(*Channel_43*)
	aPage_Channel[43].PARAM_NAME := 'Channel_43_ENC04';
	aPage_Channel[43].PARAM_00   := 4;
	aPage_Channel[43].PARAM_01   := 400;
	aPage_Channel[43].PARAM_02   := 0;
	aPage_Channel[43].PARAM_03   := 0;
	aPage_Channel[43].PARAM_04   := 0;
	aPage_Channel[43].PARAM_05   := 0;
	aPage_Channel[43].PARAM_06   := 0;
	aPage_Channel[43].PARAM_07   := 0;
	aPage_Channel[43].PARAM_08   := 0;
	aPage_Channel[43].PARAM_09   := 4;
	aPage_Channel[43].PARAM_10   := 0;

(*Channel_44*)
	aPage_Channel[44].PARAM_NAME := 'Channel_44_ENC05';
	aPage_Channel[44].PARAM_00   := 4;
	aPage_Channel[44].PARAM_01   := 500;
	aPage_Channel[44].PARAM_02   := 0;
	aPage_Channel[44].PARAM_03   := 0;
	aPage_Channel[44].PARAM_04   := 0;
	aPage_Channel[44].PARAM_05   := 0;
	aPage_Channel[44].PARAM_06   := 0;
	aPage_Channel[44].PARAM_07   := 0;
	aPage_Channel[44].PARAM_08   := 0;
	aPage_Channel[44].PARAM_09   := 5;
	aPage_Channel[44].PARAM_10   := 0;

(*Channel_45*)
	aPage_Channel[45].PARAM_NAME := 'Channel_45_ENC06';
	aPage_Channel[45].PARAM_00   := 4;
	aPage_Channel[45].PARAM_01   := 600;
	aPage_Channel[45].PARAM_02   := 0;
	aPage_Channel[45].PARAM_03   := 0;
	aPage_Channel[45].PARAM_04   := 0;
	aPage_Channel[45].PARAM_05   := 0;
	aPage_Channel[45].PARAM_06   := 0;
	aPage_Channel[45].PARAM_07   := 0;
	aPage_Channel[45].PARAM_08   := 0;
	aPage_Channel[45].PARAM_09   := 6;
	aPage_Channel[45].PARAM_10   := 0;

(*Channel_46*)
	aPage_Channel[46].PARAM_NAME := 'Channel_46_ENC07';
	aPage_Channel[46].PARAM_00   := 4;
	aPage_Channel[46].PARAM_01   := 700;
	aPage_Channel[46].PARAM_02   := 0;
	aPage_Channel[46].PARAM_03   := 0;
	aPage_Channel[46].PARAM_04   := 0;
	aPage_Channel[46].PARAM_05   := 0;
	aPage_Channel[46].PARAM_06   := 0;
	aPage_Channel[46].PARAM_07   := 0;
	aPage_Channel[46].PARAM_08   := 0;
	aPage_Channel[46].PARAM_09   := 7;
	aPage_Channel[46].PARAM_10   := 0;

(*Channel_47*)
	aPage_Channel[47].PARAM_NAME := 'Channel_47_ENC08';
	aPage_Channel[47].PARAM_00   := 4;
	aPage_Channel[47].PARAM_01   := 800;
	aPage_Channel[47].PARAM_02   := 0;
	aPage_Channel[47].PARAM_03   := 0;
	aPage_Channel[47].PARAM_04   := 0;
	aPage_Channel[47].PARAM_05   := 0;
	aPage_Channel[47].PARAM_06   := 0;
	aPage_Channel[47].PARAM_07   := 0;
	aPage_Channel[47].PARAM_08   := 0;
	aPage_Channel[47].PARAM_09   := 8;
	aPage_Channel[47].PARAM_10   := 0;

(*Channel_48*)
	aPage_Channel[48].PARAM_NAME := 'Channel_48_FRM01';
	aPage_Channel[48].PARAM_00   := 5;
	aPage_Channel[48].PARAM_01   := 1;
	aPage_Channel[48].PARAM_02   := 2;
	aPage_Channel[48].PARAM_03   := 3;
	aPage_Channel[48].PARAM_04   := 4;
	aPage_Channel[48].PARAM_05   := 5;
	aPage_Channel[48].PARAM_06   := 0;
	aPage_Channel[48].PARAM_07   := 0;
	aPage_Channel[48].PARAM_08   := 0;
	aPage_Channel[48].PARAM_09   := 1;
	aPage_Channel[48].PARAM_10   := 0;

(*Channel_49*)
	aPage_Channel[49].PARAM_NAME := 'Channel_49_FRM02';
	aPage_Channel[49].PARAM_00   := 5;
	aPage_Channel[49].PARAM_01   := 1;
	aPage_Channel[49].PARAM_02   := 2;
	aPage_Channel[49].PARAM_03   := 3;
	aPage_Channel[49].PARAM_04   := 4;
	aPage_Channel[49].PARAM_05   := 5;
	aPage_Channel[49].PARAM_06   := 0;
	aPage_Channel[49].PARAM_07   := 0;
	aPage_Channel[49].PARAM_08   := 0;
	aPage_Channel[49].PARAM_09   := 2;
	aPage_Channel[49].PARAM_10   := 0;

(*Channel_50*)
	aPage_Channel[50].PARAM_NAME := 'Channel_50_FRM03';
	aPage_Channel[50].PARAM_00   := 5;
	aPage_Channel[50].PARAM_01   := 1;
	aPage_Channel[50].PARAM_02   := 2;
	aPage_Channel[50].PARAM_03   := 3;
	aPage_Channel[50].PARAM_04   := 4;
	aPage_Channel[50].PARAM_05   := 5;
	aPage_Channel[50].PARAM_06   := 0;
	aPage_Channel[50].PARAM_07   := 0;
	aPage_Channel[50].PARAM_08   := 0;
	aPage_Channel[50].PARAM_09   := 3;
	aPage_Channel[50].PARAM_10   := 0;

(*Channel_51*)
	aPage_Channel[51].PARAM_NAME := 'Channel_51_FRM04';
	aPage_Channel[51].PARAM_00   := 5;
	aPage_Channel[51].PARAM_01   := 1;
	aPage_Channel[51].PARAM_02   := 2;
	aPage_Channel[51].PARAM_03   := 3;
	aPage_Channel[51].PARAM_04   := 4;
	aPage_Channel[51].PARAM_05   := 5;
	aPage_Channel[51].PARAM_06   := 0;
	aPage_Channel[51].PARAM_07   := 0;
	aPage_Channel[51].PARAM_08   := 0;
	aPage_Channel[51].PARAM_09   := 4;
	aPage_Channel[51].PARAM_10   := 0;

(*Channel_52*)
	aPage_Channel[52].PARAM_NAME := 'Channel_52_FRM05';
	aPage_Channel[52].PARAM_00   := 5;
	aPage_Channel[52].PARAM_01   := 1;
	aPage_Channel[52].PARAM_02   := 2;
	aPage_Channel[52].PARAM_03   := 3;
	aPage_Channel[52].PARAM_04   := 4;
	aPage_Channel[52].PARAM_05   := 5;
	aPage_Channel[52].PARAM_06   := 0;
	aPage_Channel[52].PARAM_07   := 0;
	aPage_Channel[52].PARAM_08   := 0;
	aPage_Channel[52].PARAM_09   := 5;
	aPage_Channel[52].PARAM_10   := 0;

(*Channel_53*)
	aPage_Channel[53].PARAM_NAME := 'Channel_53_FRM06';
	aPage_Channel[53].PARAM_00   := 5;
	aPage_Channel[53].PARAM_01   := 1;
	aPage_Channel[53].PARAM_02   := 2;
	aPage_Channel[53].PARAM_03   := 3;
	aPage_Channel[53].PARAM_04   := 4;
	aPage_Channel[53].PARAM_05   := 5;
	aPage_Channel[53].PARAM_06   := 0;
	aPage_Channel[53].PARAM_07   := 0;
	aPage_Channel[53].PARAM_08   := 0;
	aPage_Channel[53].PARAM_09   := 6;
	aPage_Channel[53].PARAM_10   := 0;

(*Channel_54*)
	aPage_Channel[54].PARAM_NAME := 'Channel_54_FRM07';
	aPage_Channel[54].PARAM_00   := 5;
	aPage_Channel[54].PARAM_01   := 1;
	aPage_Channel[54].PARAM_02   := 2;
	aPage_Channel[54].PARAM_03   := 3;
	aPage_Channel[54].PARAM_04   := 4;
	aPage_Channel[54].PARAM_05   := 5;
	aPage_Channel[54].PARAM_06   := 0;
	aPage_Channel[54].PARAM_07   := 0;
	aPage_Channel[54].PARAM_08   := 0;
	aPage_Channel[54].PARAM_09   := 7;
	aPage_Channel[54].PARAM_10   := 0;

(*Channel_55*)
	aPage_Channel[55].PARAM_NAME := 'Channel_55_FRM08';
	aPage_Channel[55].PARAM_00   := 5;
	aPage_Channel[55].PARAM_01   := 1;
	aPage_Channel[55].PARAM_02   := 2;
	aPage_Channel[55].PARAM_03   := 3;
	aPage_Channel[55].PARAM_04   := 4;
	aPage_Channel[55].PARAM_05   := 5;
	aPage_Channel[55].PARAM_06   := 0;
	aPage_Channel[55].PARAM_07   := 0;
	aPage_Channel[55].PARAM_08   := 0;
	aPage_Channel[55].PARAM_09   := 8;
	aPage_Channel[55].PARAM_10   := 0;

(*Channel_56*)
	aPage_Channel[56].PARAM_NAME := 'Channel_56_SPR01';
	aPage_Channel[56].PARAM_00   := 6;
	aPage_Channel[56].PARAM_01   := 1;
	aPage_Channel[56].PARAM_02   := 1;
	aPage_Channel[56].PARAM_03   := 1;
	aPage_Channel[56].PARAM_04   := 1;
	aPage_Channel[56].PARAM_05   := 1;
	aPage_Channel[56].PARAM_06   := 0;
	aPage_Channel[56].PARAM_07   := 0;
	aPage_Channel[56].PARAM_08   := 0;
	aPage_Channel[56].PARAM_09   := 1;
	aPage_Channel[56].PARAM_10   := 0;

(*Channel_57*)
	aPage_Channel[57].PARAM_NAME := 'Channel_57_SPR02';
	aPage_Channel[57].PARAM_00   := 6;
	aPage_Channel[57].PARAM_01   := 1;
	aPage_Channel[57].PARAM_02   := 1;
	aPage_Channel[57].PARAM_03   := 1;
	aPage_Channel[57].PARAM_04   := 1;
	aPage_Channel[57].PARAM_05   := 1;
	aPage_Channel[57].PARAM_06   := 0;
	aPage_Channel[57].PARAM_07   := 0;
	aPage_Channel[57].PARAM_08   := 0;
	aPage_Channel[57].PARAM_09   := 2;
	aPage_Channel[57].PARAM_10   := 0;

(*Channel_58*)
	aPage_Channel[58].PARAM_NAME := 'Channel_58_SPR03';
	aPage_Channel[58].PARAM_00   := 6;
	aPage_Channel[58].PARAM_01   := 1;
	aPage_Channel[58].PARAM_02   := 1;
	aPage_Channel[58].PARAM_03   := 1;
	aPage_Channel[58].PARAM_04   := 1;
	aPage_Channel[58].PARAM_05   := 1;
	aPage_Channel[58].PARAM_06   := 0;
	aPage_Channel[58].PARAM_07   := 0;
	aPage_Channel[58].PARAM_08   := 0;
	aPage_Channel[58].PARAM_09   := 3;
	aPage_Channel[58].PARAM_10   := 0;

(*Channel_59*)
	aPage_Channel[59].PARAM_NAME := 'Channel_59_SPR04';
	aPage_Channel[59].PARAM_00   := 6;
	aPage_Channel[59].PARAM_01   := 1;
	aPage_Channel[59].PARAM_02   := 1;
	aPage_Channel[59].PARAM_03   := 1;
	aPage_Channel[59].PARAM_04   := 1;
	aPage_Channel[59].PARAM_05   := 1;
	aPage_Channel[59].PARAM_06   := 0;
	aPage_Channel[59].PARAM_07   := 0;
	aPage_Channel[59].PARAM_08   := 0;
	aPage_Channel[59].PARAM_09   := 4;
	aPage_Channel[59].PARAM_10   := 0;

(*Channel_60*)
	aPage_Channel[60].PARAM_NAME := 'Channel_60_SPR05';
	aPage_Channel[60].PARAM_00   := 6;
	aPage_Channel[60].PARAM_01   := 1;
	aPage_Channel[60].PARAM_02   := 1;
	aPage_Channel[60].PARAM_03   := 1;
	aPage_Channel[60].PARAM_04   := 1;
	aPage_Channel[60].PARAM_05   := 1;
	aPage_Channel[60].PARAM_06   := 0;
	aPage_Channel[60].PARAM_07   := 0;
	aPage_Channel[60].PARAM_08   := 0;
	aPage_Channel[60].PARAM_09   := 5;
	aPage_Channel[60].PARAM_10   := 0;

(*Channel_61*)
	aPage_Channel[61].PARAM_NAME := 'Channel_61_SPR06';
	aPage_Channel[61].PARAM_00   := 6;
	aPage_Channel[61].PARAM_01   := 1;
	aPage_Channel[61].PARAM_02   := 1;
	aPage_Channel[61].PARAM_03   := 1;
	aPage_Channel[61].PARAM_04   := 1;
	aPage_Channel[61].PARAM_05   := 1;
	aPage_Channel[61].PARAM_06   := 0;
	aPage_Channel[61].PARAM_07   := 0;
	aPage_Channel[61].PARAM_08   := 0;
	aPage_Channel[61].PARAM_09   := 6;
	aPage_Channel[61].PARAM_10   := 0;

(*Channel_62*)
	aPage_Channel[62].PARAM_NAME := 'Channel_62_SPR07';
	aPage_Channel[62].PARAM_00   := 6;
	aPage_Channel[62].PARAM_01   := 1;
	aPage_Channel[62].PARAM_02   := 1;
	aPage_Channel[62].PARAM_03   := 1;
	aPage_Channel[62].PARAM_04   := 1;
	aPage_Channel[62].PARAM_05   := 1;
	aPage_Channel[62].PARAM_06   := 0;
	aPage_Channel[62].PARAM_07   := 0;
	aPage_Channel[62].PARAM_08   := 0;
	aPage_Channel[62].PARAM_09   := 7;
	aPage_Channel[62].PARAM_10   := 0;

(*Channel_63*)
	aPage_Channel[63].PARAM_NAME := 'Channel_63_SPR08';
	aPage_Channel[63].PARAM_00   := 6;
	aPage_Channel[63].PARAM_01   := 1;
	aPage_Channel[63].PARAM_02   := 1;
	aPage_Channel[63].PARAM_03   := 1;
	aPage_Channel[63].PARAM_04   := 1;
	aPage_Channel[63].PARAM_05   := 1;
	aPage_Channel[63].PARAM_06   := 0;
	aPage_Channel[63].PARAM_07   := 0;
	aPage_Channel[63].PARAM_08   := 0;
	aPage_Channel[63].PARAM_09   := 8;
	aPage_Channel[63].PARAM_10   := 0;

(*-----------------------------------------------------------------------------------------------------------------------------------------------------------------------------------*)
(**)

	DefaultSettingsTestModeRecovery;

	bCurrModeChange := 0;

END_IF;
END_PROGRAM

(* POU Default_Settings/FLASH_TO_PAGE_CHANNEL, ST *)
FUNCTION_BLOCK FLASH_TO_PAGE_CHANNEL

VAR_INPUT
	bInit         : BOOL;
END_VAR

VAR_OUTPUT
END_VAR

VAR
	instFRAMWrite : FRAMWRITE;
	i             : INT := 0;
END_VAR
(*-----------------------------------------------------------------------------------------------------------------------------------------------------------------------------------*)
(*Запись в энергонезависимую память установочных параметров, коэффициентов*)

FOR i := 0 TO 63 DO
	instFRAMWrite(Enable := 1, DST := iMemAdrArrayParamName + i * 32, LEN := 32, SRC := ADR(aPage_Channel[i].PARAM_NAME));

	instFRAMWrite(Enable := 1, DST := iMemAdrArrayParam00 + i * 4,    LEN := 4,  SRC := ADR(aPage_Channel[i].PARAM_00));
	instFRAMWrite(Enable := 1, DST := iMemAdrArrayParam01 + i * 4,    LEN := 4,  SRC := ADR(aPage_Channel[i].PARAM_01));
	instFRAMWrite(Enable := 1, DST := iMemAdrArrayParam02 + i * 4,    LEN := 4,  SRC := ADR(aPage_Channel[i].PARAM_02));
	instFRAMWrite(Enable := 1, DST := iMemAdrArrayParam03 + i * 4,    LEN := 4,  SRC := ADR(aPage_Channel[i].PARAM_03));
	instFRAMWrite(Enable := 1, DST := iMemAdrArrayParam04 + i * 4,    LEN := 4,  SRC := ADR(aPage_Channel[i].PARAM_04));
	instFRAMWrite(Enable := 1, DST := iMemAdrArrayParam05 + i * 4,    LEN := 4,  SRC := ADR(aPage_Channel[i].PARAM_05));
	instFRAMWrite(Enable := 1, DST := iMemAdrArrayParam06 + i * 4,    LEN := 4,  SRC := ADR(aPage_Channel[i].PARAM_06));
	instFRAMWrite(Enable := 1, DST := iMemAdrArrayParam07 + i * 4,    LEN := 4,  SRC := ADR(aPage_Channel[i].PARAM_07));

	instFRAMWrite(Enable := 1, DST := iMemAdrArrayParam09 + i * 4,    LEN := 4,  SRC := ADR(aPage_Channel[i].PARAM_09));
	instFRAMWrite(Enable := 1, DST := iMemAdrArrayParam10 + i * 4,    LEN := 4,  SRC := ADR(aPage_Channel[i].PARAM_10));
END_FOR;
END_FUNCTION_BLOCK

(* POU Default_Settings/Default_Settings_UnitMode_processing, ST *)
PROGRAM Default_Settings_UnitMode_processing

VAR_INPUT
	bInit                           : BOOL;
END_VAR

VAR
	DefaultSettingsUnitModeRecovery : FLASH_TO_PAGE_CHANNEL;
END_VAR
(*-----------------------------------------------------------------------------------------------------------------------------------------------------------------------------------*)
(*Восстановление заводских установок*)

IF bCurrModeChange = 1 AND dwCurrMode = 1 THEN

(*Channel_00*)
	aPage_Channel[00].PARAM_NAME := 'Давл. подпитки';
	aPage_Channel[00].PARAM_00   := 0;
	aPage_Channel[00].PARAM_01   := 3259;
	aPage_Channel[00].PARAM_02   := 648;
	aPage_Channel[00].PARAM_03   := 1.6 (*1.378951*);(*МПа, = 200 PSI*)
	aPage_Channel[00].PARAM_04   := 0;
	aPage_Channel[00].PARAM_05   := 100;
	aPage_Channel[00].PARAM_06   := 0;
	aPage_Channel[00].PARAM_07   := 0;
	aPage_Channel[00].PARAM_08   := 0;
	aPage_Channel[00].PARAM_09   := 1;
	aPage_Channel[00].PARAM_10   := 0;

(*Channel_01*)
	aPage_Channel[01].PARAM_NAME := 'Темп. азота жидкого';
	aPage_Channel[01].PARAM_00   := 0;
	aPage_Channel[01].PARAM_01   := 3259;
	aPage_Channel[01].PARAM_02   := 648;
	aPage_Channel[01].PARAM_03   := 76.666667;(*C, = 170 F*)
	aPage_Channel[01].PARAM_04   :=-195.555556;(*C, = 320 F*)
	aPage_Channel[01].PARAM_05   := 100;
	aPage_Channel[01].PARAM_06   := 0;
	aPage_Channel[01].PARAM_07   := 0;
	aPage_Channel[01].PARAM_08   := 0;
	aPage_Channel[01].PARAM_09   := 2;
	aPage_Channel[01].PARAM_10   := 0;

(*Channel_02*)
	aPage_Channel[02].PARAM_NAME := 'Темп. нагнетания';
	aPage_Channel[02].PARAM_00   := 0;
	aPage_Channel[02].PARAM_01   := 3259;
	aPage_Channel[02].PARAM_02   := 648;
	aPage_Channel[02].PARAM_03   := 50;
	aPage_Channel[02].PARAM_04   :=-50;
	aPage_Channel[02].PARAM_05   := 100;
	aPage_Channel[02].PARAM_06   := 0;
	aPage_Channel[02].PARAM_07   := 0;
	aPage_Channel[02].PARAM_08   := 0;
	aPage_Channel[02].PARAM_09   := 4;
	aPage_Channel[02].PARAM_10   := 0;

(*Channel_03*)
	aPage_Channel[03].PARAM_NAME := 'Давл. нагнетания';
	aPage_Channel[03].PARAM_00   := 0;
	aPage_Channel[03].PARAM_01   := 3259;
	aPage_Channel[03].PARAM_02   := 648;
	aPage_Channel[03].PARAM_03   := 103.421351;(*МПа, = 15000 PSI*)
	aPage_Channel[03].PARAM_04   := 0;
	aPage_Channel[03].PARAM_05   := 100;
	aPage_Channel[03].PARAM_06   := 0;
	aPage_Channel[03].PARAM_07   := 0;
	aPage_Channel[03].PARAM_08   := 0;
	aPage_Channel[03].PARAM_09   := 5;
	aPage_Channel[03].PARAM_10   := 0;

(*Channel_04*)
	aPage_Channel[04].PARAM_NAME := 'Давл. гидронагрева';
	aPage_Channel[04].PARAM_00   := 0;
	aPage_Channel[04].PARAM_01   := 3259;
	aPage_Channel[04].PARAM_02   := 648;
	aPage_Channel[04].PARAM_03   := 40;
	aPage_Channel[04].PARAM_04   := 0;
	aPage_Channel[04].PARAM_05   := 100;
	aPage_Channel[04].PARAM_06   := 0;
	aPage_Channel[04].PARAM_07   := 0;
	aPage_Channel[04].PARAM_08   := 0;
	aPage_Channel[04].PARAM_09   := 6;
	aPage_Channel[04].PARAM_10   := 0;

(*Channel_05*)
	aPage_Channel[05].PARAM_NAME := 'Темп. ОЖ до испарителя';
	aPage_Channel[05].PARAM_00   := 0;
	aPage_Channel[05].PARAM_01   := 3259;
	aPage_Channel[05].PARAM_02   := 648;
	aPage_Channel[05].PARAM_03   := 150;
	aPage_Channel[05].PARAM_04   :=-50;
	aPage_Channel[05].PARAM_05   := 100;
	aPage_Channel[05].PARAM_06   := 0;
	aPage_Channel[05].PARAM_07   := 0;
	aPage_Channel[05].PARAM_08   := 0;
	aPage_Channel[05].PARAM_09   := 3;
	aPage_Channel[05].PARAM_10   := 0;

(*Channel_06*)
	aPage_Channel[06].PARAM_NAME := 'Обороты НВД';
	aPage_Channel[06].PARAM_00   := 1;
	aPage_Channel[06].PARAM_01   := 8_200;
	aPage_Channel[06].PARAM_02   := 0;
	aPage_Channel[06].PARAM_03   := 6_000;
	aPage_Channel[06].PARAM_04   := 0;
	aPage_Channel[06].PARAM_05   := 1_000;
	aPage_Channel[06].PARAM_06   := 0;
	aPage_Channel[06].PARAM_07   := 0;
	aPage_Channel[06].PARAM_08   := 0;
	aPage_Channel[06].PARAM_09   := 1;
	aPage_Channel[06].PARAM_10   := 0;

(*Channel_07*)
	aPage_Channel[07].PARAM_NAME := 'Давл. гидронагрева';
	aPage_Channel[07].PARAM_00   := 2;
	aPage_Channel[07].PARAM_01   := 100;
	aPage_Channel[07].PARAM_02   := 0;
	aPage_Channel[07].PARAM_03   := 540 (*500*);
	aPage_Channel[07].PARAM_04   := 0;
	aPage_Channel[07].PARAM_05   := 4_000;
	aPage_Channel[07].PARAM_06   := 0;
	aPage_Channel[07].PARAM_07   := 0;
	aPage_Channel[07].PARAM_08   := 0;
	aPage_Channel[07].PARAM_09   := 1;
	aPage_Channel[07].PARAM_10   := 0;

(*Channel_08*)
	aPage_Channel[08].PARAM_NAME := 'Обороты НВД';
	aPage_Channel[08].PARAM_00   := 2;
	aPage_Channel[08].PARAM_01   := 100;
	aPage_Channel[08].PARAM_02   := 0;
	aPage_Channel[08].PARAM_03   := 460 (*400*);
	aPage_Channel[08].PARAM_04   := 0;
	aPage_Channel[08].PARAM_05   := 4_000;
	aPage_Channel[08].PARAM_06   := 0;
	aPage_Channel[08].PARAM_07   := 0;
	aPage_Channel[08].PARAM_08   := 0;
	aPage_Channel[08].PARAM_09   := 2;
	aPage_Channel[08].PARAM_10   := 0;

(*Channel_09*)
	aPage_Channel[09].PARAM_NAME := 'Давл. подпитки';
	aPage_Channel[09].PARAM_00   := 2;
	aPage_Channel[09].PARAM_01   := 100;
	aPage_Channel[09].PARAM_02   := 0;
	aPage_Channel[09].PARAM_03   := 400;
	aPage_Channel[09].PARAM_04   := 0;
	aPage_Channel[09].PARAM_05   := 4_000;
	aPage_Channel[09].PARAM_06   := 0;
	aPage_Channel[09].PARAM_07   := 0;
	aPage_Channel[09].PARAM_08   := 0;
	aPage_Channel[09].PARAM_09   := 3;
	aPage_Channel[09].PARAM_10   := 0;

(*Channel_10*)
	aPage_Channel[10].PARAM_NAME := 'Давл. гидронагрева';
	aPage_Channel[10].PARAM_00   := 3;
	aPage_Channel[10].PARAM_01   := 20 (*250*);
	aPage_Channel[10].PARAM_02   := 50;
	aPage_Channel[10].PARAM_03   := 0;
	aPage_Channel[10].PARAM_04   := 0;
	aPage_Channel[10].PARAM_05   := 0;
	aPage_Channel[10].PARAM_06   := 0;
	aPage_Channel[10].PARAM_07   := 0;
	aPage_Channel[10].PARAM_08   := 0;
	aPage_Channel[10].PARAM_09   := 1;
	aPage_Channel[10].PARAM_10   := 0;

(*Channel_11*)
	aPage_Channel[11].PARAM_NAME := 'Обороты НВД';
	aPage_Channel[11].PARAM_00   := 3;
	aPage_Channel[11].PARAM_01   := 0.001 (*0.005*);
	aPage_Channel[11].PARAM_02   := 0.05;
	aPage_Channel[11].PARAM_03   := 0;
	aPage_Channel[11].PARAM_04   := 180;
	aPage_Channel[11].PARAM_05   := 0;
	aPage_Channel[11].PARAM_06   := 0;
	aPage_Channel[11].PARAM_07   := 0;
	aPage_Channel[11].PARAM_08   := 0;
	aPage_Channel[11].PARAM_09   := 2;
	aPage_Channel[11].PARAM_10   := 0;

(*Channel_12*)
	aPage_Channel[12].PARAM_NAME := 'Давл. подпитки';
	aPage_Channel[12].PARAM_00   := 3;
	aPage_Channel[12].PARAM_01   := 30 (*80*);
	aPage_Channel[12].PARAM_02   := 0.250;
	aPage_Channel[12].PARAM_03   := 0;
	aPage_Channel[12].PARAM_04   := 0;
	aPage_Channel[12].PARAM_05   := 0;
	aPage_Channel[12].PARAM_06   := 0;
	aPage_Channel[12].PARAM_07   := 0;
	aPage_Channel[12].PARAM_08   := 0;
	aPage_Channel[12].PARAM_09   := 3;
	aPage_Channel[12].PARAM_10   := 0;

(*Channel_13*)
	aPage_Channel[13].PARAM_NAME := 'Channel_13';
	aPage_Channel[13].PARAM_00   := 9;
	aPage_Channel[13].PARAM_01   := 1;
	aPage_Channel[13].PARAM_02   := 1;
	aPage_Channel[13].PARAM_03   := 1;
	aPage_Channel[13].PARAM_04   := 1;
	aPage_Channel[13].PARAM_05   := 1;
	aPage_Channel[13].PARAM_06   := 0;
	aPage_Channel[13].PARAM_07   := 0;
	aPage_Channel[13].PARAM_08   := 0;
	aPage_Channel[13].PARAM_09   := 0;
	aPage_Channel[13].PARAM_10   := 0;

(*Channel_14*)
	aPage_Channel[14].PARAM_NAME := 'Channel_14';
	aPage_Channel[14].PARAM_00   := 9;
	aPage_Channel[14].PARAM_01   := 1;
	aPage_Channel[14].PARAM_02   := 1;
	aPage_Channel[14].PARAM_03   := 1;
	aPage_Channel[14].PARAM_04   := 1;
	aPage_Channel[14].PARAM_05   := 1;
	aPage_Channel[14].PARAM_06   := 0;
	aPage_Channel[14].PARAM_07   := 0;
	aPage_Channel[14].PARAM_08   := 0;
	aPage_Channel[14].PARAM_09   := 0;
	aPage_Channel[14].PARAM_10   := 0;

(*Channel_15*)
	aPage_Channel[15].PARAM_NAME := 'Channel_15';
	aPage_Channel[15].PARAM_00   := 9;
	aPage_Channel[15].PARAM_01   := 1;
	aPage_Channel[15].PARAM_02   := 1;
	aPage_Channel[15].PARAM_03   := 1;
	aPage_Channel[15].PARAM_04   := 1;
	aPage_Channel[15].PARAM_05   := 1;
	aPage_Channel[15].PARAM_06   := 0;
	aPage_Channel[15].PARAM_07   := 0;
	aPage_Channel[15].PARAM_08   := 0;
	aPage_Channel[15].PARAM_09   := 0;
	aPage_Channel[15].PARAM_10   := 0;

(*Channel_16*)
	aPage_Channel[16].PARAM_NAME := 'Channel_16';
	aPage_Channel[16].PARAM_00   := 9;
	aPage_Channel[16].PARAM_01   := 1;
	aPage_Channel[16].PARAM_02   := 1;
	aPage_Channel[16].PARAM_03   := 1;
	aPage_Channel[16].PARAM_04   := 1;
	aPage_Channel[16].PARAM_05   := 1;
	aPage_Channel[16].PARAM_06   := 0;
	aPage_Channel[16].PARAM_07   := 0;
	aPage_Channel[16].PARAM_08   := 0;
	aPage_Channel[16].PARAM_09   := 0;
	aPage_Channel[16].PARAM_10   := 0;

(*Channel_17*)
	aPage_Channel[17].PARAM_NAME := 'Channel_17';
	aPage_Channel[17].PARAM_00   := 9;
	aPage_Channel[17].PARAM_01   := 1;
	aPage_Channel[17].PARAM_02   := 1;
	aPage_Channel[17].PARAM_03   := 1;
	aPage_Channel[17].PARAM_04   := 1;
	aPage_Channel[17].PARAM_05   := 1;
	aPage_Channel[17].PARAM_06   := 0;
	aPage_Channel[17].PARAM_07   := 0;
	aPage_Channel[17].PARAM_08   := 0;
	aPage_Channel[17].PARAM_09   := 0;
	aPage_Channel[17].PARAM_10   := 0;

(*Channel_18*)
	aPage_Channel[18].PARAM_NAME := 'Channel_18';
	aPage_Channel[18].PARAM_00   := 9;
	aPage_Channel[18].PARAM_01   := 1;
	aPage_Channel[18].PARAM_02   := 1;
	aPage_Channel[18].PARAM_03   := 1;
	aPage_Channel[18].PARAM_04   := 1;
	aPage_Channel[18].PARAM_05   := 1;
	aPage_Channel[18].PARAM_06   := 0;
	aPage_Channel[18].PARAM_07   := 0;
	aPage_Channel[18].PARAM_08   := 0;
	aPage_Channel[18].PARAM_09   := 0;
	aPage_Channel[18].PARAM_10   := 0;

(*Channel_19*)
	aPage_Channel[19].PARAM_NAME := 'Channel_19';
	aPage_Channel[19].PARAM_00   := 9;
	aPage_Channel[19].PARAM_01   := 1;
	aPage_Channel[19].PARAM_02   := 1;
	aPage_Channel[19].PARAM_03   := 1;
	aPage_Channel[19].PARAM_04   := 1;
	aPage_Channel[19].PARAM_05   := 1;
	aPage_Channel[19].PARAM_06   := 0;
	aPage_Channel[19].PARAM_07   := 0;
	aPage_Channel[19].PARAM_08   := 0;
	aPage_Channel[19].PARAM_09   := 0;
	aPage_Channel[19].PARAM_10   := 0;

(*Channel_20*)
	aPage_Channel[20].PARAM_NAME := 'Channel_20';
	aPage_Channel[20].PARAM_00   := 9;
	aPage_Channel[20].PARAM_01   := 1;
	aPage_Channel[20].PARAM_02   := 1;
	aPage_Channel[20].PARAM_03   := 1;
	aPage_Channel[20].PARAM_04   := 1;
	aPage_Channel[20].PARAM_05   := 1;
	aPage_Channel[20].PARAM_06   := 0;
	aPage_Channel[20].PARAM_07   := 0;
	aPage_Channel[20].PARAM_08   := 0;
	aPage_Channel[20].PARAM_09   := 0;
	aPage_Channel[20].PARAM_10   := 0;

(*Channel_21*)
	aPage_Channel[21].PARAM_NAME := 'Channel_21';
	aPage_Channel[21].PARAM_00   := 9;
	aPage_Channel[21].PARAM_01   := 1;
	aPage_Channel[21].PARAM_02   := 1;
	aPage_Channel[21].PARAM_03   := 1;
	aPage_Channel[21].PARAM_04   := 1;
	aPage_Channel[21].PARAM_05   := 1;
	aPage_Channel[21].PARAM_06   := 0;
	aPage_Channel[21].PARAM_07   := 0;
	aPage_Channel[21].PARAM_08   := 0;
	aPage_Channel[21].PARAM_09   := 0;
	aPage_Channel[21].PARAM_10   := 0;

(*Channel_22*)
	aPage_Channel[22].PARAM_NAME := 'Channel_22';
	aPage_Channel[22].PARAM_00   := 9;
	aPage_Channel[22].PARAM_01   := 1;
	aPage_Channel[22].PARAM_02   := 1;
	aPage_Channel[22].PARAM_03   := 1;
	aPage_Channel[22].PARAM_04   := 1;
	aPage_Channel[22].PARAM_05   := 1;
	aPage_Channel[22].PARAM_06   := 0;
	aPage_Channel[22].PARAM_07   := 0;
	aPage_Channel[22].PARAM_08   := 0;
	aPage_Channel[22].PARAM_09   := 0;
	aPage_Channel[22].PARAM_10   := 0;

(*Channel_23*)
	aPage_Channel[23].PARAM_NAME := 'Channel_23';
	aPage_Channel[23].PARAM_00   := 9;
	aPage_Channel[23].PARAM_01   := 1;
	aPage_Channel[23].PARAM_02   := 1;
	aPage_Channel[23].PARAM_03   := 1;
	aPage_Channel[23].PARAM_04   := 1;
	aPage_Channel[23].PARAM_05   := 1;
	aPage_Channel[23].PARAM_06   := 0;
	aPage_Channel[23].PARAM_07   := 0;
	aPage_Channel[23].PARAM_08   := 0;
	aPage_Channel[23].PARAM_09   := 0;
	aPage_Channel[23].PARAM_10   := 0;

(*Channel_24*)
	aPage_Channel[24].PARAM_NAME := 'Channel_24';
	aPage_Channel[24].PARAM_00   := 9;
	aPage_Channel[24].PARAM_01   := 1;
	aPage_Channel[24].PARAM_02   := 1;
	aPage_Channel[24].PARAM_03   := 1;
	aPage_Channel[24].PARAM_04   := 1;
	aPage_Channel[24].PARAM_05   := 1;
	aPage_Channel[24].PARAM_06   := 0;
	aPage_Channel[24].PARAM_07   := 0;
	aPage_Channel[24].PARAM_08   := 0;
	aPage_Channel[24].PARAM_09   := 0;
	aPage_Channel[24].PARAM_10   := 0;

(*Channel_25*)
	aPage_Channel[25].PARAM_NAME := 'Channel_25';
	aPage_Channel[25].PARAM_00   := 9;
	aPage_Channel[25].PARAM_01   := 1;
	aPage_Channel[25].PARAM_02   := 1;
	aPage_Channel[25].PARAM_03   := 1;
	aPage_Channel[25].PARAM_04   := 1;
	aPage_Channel[25].PARAM_05   := 1;
	aPage_Channel[25].PARAM_06   := 0;
	aPage_Channel[25].PARAM_07   := 0;
	aPage_Channel[25].PARAM_08   := 0;
	aPage_Channel[25].PARAM_09   := 0;
	aPage_Channel[25].PARAM_10   := 0;

(*Channel_26*)
	aPage_Channel[26].PARAM_NAME := 'Channel_26';
	aPage_Channel[26].PARAM_00   := 9;
	aPage_Channel[26].PARAM_01   := 1;
	aPage_Channel[26].PARAM_02   := 1;
	aPage_Channel[26].PARAM_03   := 1;
	aPage_Channel[26].PARAM_04   := 1;
	aPage_Channel[26].PARAM_05   := 1;
	aPage_Channel[26].PARAM_06   := 0;
	aPage_Channel[26].PARAM_07   := 0;
	aPage_Channel[26].PARAM_08   := 0;
	aPage_Channel[26].PARAM_09   := 0;
	aPage_Channel[26].PARAM_10   := 0;

(*Channel_27*)
	aPage_Channel[27].PARAM_NAME := 'Channel_27';
	aPage_Channel[27].PARAM_00   := 9;
	aPage_Channel[27].PARAM_01   := 1;
	aPage_Channel[27].PARAM_02   := 1;
	aPage_Channel[27].PARAM_03   := 1;
	aPage_Channel[27].PARAM_04   := 1;
	aPage_Channel[27].PARAM_05   := 1;
	aPage_Channel[27].PARAM_06   := 0;
	aPage_Channel[27].PARAM_07   := 0;
	aPage_Channel[27].PARAM_08   := 0;
	aPage_Channel[27].PARAM_09   := 0;
	aPage_Channel[27].PARAM_10   := 0;

(*Channel_28*)
	aPage_Channel[28].PARAM_NAME := 'Channel_28';
	aPage_Channel[28].PARAM_00   := 9;
	aPage_Channel[28].PARAM_01   := 1;
	aPage_Channel[28].PARAM_02   := 1;
	aPage_Channel[28].PARAM_03   := 1;
	aPage_Channel[28].PARAM_04   := 1;
	aPage_Channel[28].PARAM_05   := 1;
	aPage_Channel[28].PARAM_06   := 0;
	aPage_Channel[28].PARAM_07   := 0;
	aPage_Channel[28].PARAM_08   := 0;
	aPage_Channel[28].PARAM_09   := 0;
	aPage_Channel[28].PARAM_10   := 0;

(*Channel_29*)
	aPage_Channel[29].PARAM_NAME := 'Channel_29';
	aPage_Channel[29].PARAM_00   := 9;
	aPage_Channel[29].PARAM_01   := 1;
	aPage_Channel[29].PARAM_02   := 1;
	aPage_Channel[29].PARAM_03   := 1;
	aPage_Channel[29].PARAM_04   := 1;
	aPage_Channel[29].PARAM_05   := 1;
	aPage_Channel[29].PARAM_06   := 0;
	aPage_Channel[29].PARAM_07   := 0;
	aPage_Channel[29].PARAM_08   := 0;
	aPage_Channel[29].PARAM_09   := 0;
	aPage_Channel[29].PARAM_10   := 0;

(*Channel_30*)
	aPage_Channel[30].PARAM_NAME := 'Channel_30';
	aPage_Channel[30].PARAM_00   := 9;
	aPage_Channel[30].PARAM_01   := 1;
	aPage_Channel[30].PARAM_02   := 1;
	aPage_Channel[30].PARAM_03   := 1;
	aPage_Channel[30].PARAM_04   := 1;
	aPage_Channel[30].PARAM_05   := 1;
	aPage_Channel[30].PARAM_06   := 0;
	aPage_Channel[30].PARAM_07   := 0;
	aPage_Channel[30].PARAM_08   := 0;
	aPage_Channel[30].PARAM_09   := 0;
	aPage_Channel[30].PARAM_10   := 0;

(*Channel_31*)
	aPage_Channel[31].PARAM_NAME := 'Channel_31';
	aPage_Channel[31].PARAM_00   := 9;
	aPage_Channel[31].PARAM_01   := 1;
	aPage_Channel[31].PARAM_02   := 1;
	aPage_Channel[31].PARAM_03   := 1;
	aPage_Channel[31].PARAM_04   := 1;
	aPage_Channel[31].PARAM_05   := 1;
	aPage_Channel[31].PARAM_06   := 0;
	aPage_Channel[31].PARAM_07   := 0;
	aPage_Channel[31].PARAM_08   := 0;
	aPage_Channel[31].PARAM_09   := 0;
	aPage_Channel[31].PARAM_10   := 0;

(*Channel_32*)
	aPage_Channel[32].PARAM_NAME := 'Channel_32';
	aPage_Channel[32].PARAM_00   := 9;
	aPage_Channel[32].PARAM_01   := 1;
	aPage_Channel[32].PARAM_02   := 1;
	aPage_Channel[32].PARAM_03   := 1;
	aPage_Channel[32].PARAM_04   := 1;
	aPage_Channel[32].PARAM_05   := 1;
	aPage_Channel[32].PARAM_06   := 0;
	aPage_Channel[32].PARAM_07   := 0;
	aPage_Channel[32].PARAM_08   := 0;
	aPage_Channel[32].PARAM_09   := 0;
	aPage_Channel[32].PARAM_10   := 0;

(*Channel_33*)
	aPage_Channel[33].PARAM_NAME := 'Channel_33';
	aPage_Channel[33].PARAM_00   := 9;
	aPage_Channel[33].PARAM_01   := 1;
	aPage_Channel[33].PARAM_02   := 1;
	aPage_Channel[33].PARAM_03   := 1;
	aPage_Channel[33].PARAM_04   := 1;
	aPage_Channel[33].PARAM_05   := 1;
	aPage_Channel[33].PARAM_06   := 0;
	aPage_Channel[33].PARAM_07   := 0;
	aPage_Channel[33].PARAM_08   := 0;
	aPage_Channel[33].PARAM_09   := 0;
	aPage_Channel[33].PARAM_10   := 0;

(*Channel_34*)
	aPage_Channel[34].PARAM_NAME := 'Channel_34';
	aPage_Channel[34].PARAM_00   := 9;
	aPage_Channel[34].PARAM_01   := 1;
	aPage_Channel[34].PARAM_02   := 1;
	aPage_Channel[34].PARAM_03   := 1;
	aPage_Channel[34].PARAM_04   := 1;
	aPage_Channel[34].PARAM_05   := 1;
	aPage_Channel[34].PARAM_06   := 0;
	aPage_Channel[34].PARAM_07   := 0;
	aPage_Channel[34].PARAM_08   := 0;
	aPage_Channel[34].PARAM_09   := 0;
	aPage_Channel[34].PARAM_10   := 0;

(*Channel_35*)
	aPage_Channel[35].PARAM_NAME := 'Channel_35';
	aPage_Channel[35].PARAM_00   := 9;
	aPage_Channel[35].PARAM_01   := 1;
	aPage_Channel[35].PARAM_02   := 1;
	aPage_Channel[35].PARAM_03   := 1;
	aPage_Channel[35].PARAM_04   := 1;
	aPage_Channel[35].PARAM_05   := 1;
	aPage_Channel[35].PARAM_06   := 0;
	aPage_Channel[35].PARAM_07   := 0;
	aPage_Channel[35].PARAM_08   := 0;
	aPage_Channel[35].PARAM_09   := 0;
	aPage_Channel[35].PARAM_10   := 0;

(*Channel_36*)
	aPage_Channel[36].PARAM_NAME := 'Channel_36';
	aPage_Channel[36].PARAM_00   := 9;
	aPage_Channel[36].PARAM_01   := 1;
	aPage_Channel[36].PARAM_02   := 1;
	aPage_Channel[36].PARAM_03   := 1;
	aPage_Channel[36].PARAM_04   := 1;
	aPage_Channel[36].PARAM_05   := 1;
	aPage_Channel[36].PARAM_06   := 0;
	aPage_Channel[36].PARAM_07   := 0;
	aPage_Channel[36].PARAM_08   := 0;
	aPage_Channel[36].PARAM_09   := 0;
	aPage_Channel[36].PARAM_10   := 0;

(*Channel_37*)
	aPage_Channel[37].PARAM_NAME := 'Channel_37';
	aPage_Channel[37].PARAM_00   := 9;
	aPage_Channel[37].PARAM_01   := 1;
	aPage_Channel[37].PARAM_02   := 1;
	aPage_Channel[37].PARAM_03   := 1;
	aPage_Channel[37].PARAM_04   := 1;
	aPage_Channel[37].PARAM_05   := 1;
	aPage_Channel[37].PARAM_06   := 0;
	aPage_Channel[37].PARAM_07   := 0;
	aPage_Channel[37].PARAM_08   := 0;
	aPage_Channel[37].PARAM_09   := 0;
	aPage_Channel[37].PARAM_10   := 0;

(*Channel_38*)
	aPage_Channel[38].PARAM_NAME := 'Channel_38';
	aPage_Channel[38].PARAM_00   := 9;
	aPage_Channel[38].PARAM_01   := 1;
	aPage_Channel[38].PARAM_02   := 1;
	aPage_Channel[38].PARAM_03   := 1;
	aPage_Channel[38].PARAM_04   := 1;
	aPage_Channel[38].PARAM_05   := 1;
	aPage_Channel[38].PARAM_06   := 0;
	aPage_Channel[38].PARAM_07   := 0;
	aPage_Channel[38].PARAM_08   := 0;
	aPage_Channel[38].PARAM_09   := 0;
	aPage_Channel[38].PARAM_10   := 0;

(*Channel_39*)
	aPage_Channel[39].PARAM_NAME := 'Channel_39';
	aPage_Channel[39].PARAM_00   := 9;
	aPage_Channel[39].PARAM_01   := 1;
	aPage_Channel[39].PARAM_02   := 1;
	aPage_Channel[39].PARAM_03   := 1;
	aPage_Channel[39].PARAM_04   := 1;
	aPage_Channel[39].PARAM_05   := 1;
	aPage_Channel[39].PARAM_06   := 0;
	aPage_Channel[39].PARAM_07   := 0;
	aPage_Channel[39].PARAM_08   := 0;
	aPage_Channel[39].PARAM_09   := 0;
	aPage_Channel[39].PARAM_10   := 0;

(*Channel_40*)
	aPage_Channel[40].PARAM_NAME := 'Channel_40';
	aPage_Channel[40].PARAM_00   := 9;
	aPage_Channel[40].PARAM_01   := 1;
	aPage_Channel[40].PARAM_02   := 1;
	aPage_Channel[40].PARAM_03   := 1;
	aPage_Channel[40].PARAM_04   := 1;
	aPage_Channel[40].PARAM_05   := 1;
	aPage_Channel[40].PARAM_06   := 0;
	aPage_Channel[40].PARAM_07   := 0;
	aPage_Channel[40].PARAM_08   := 0;
	aPage_Channel[40].PARAM_09   := 0;
	aPage_Channel[40].PARAM_10   := 0;

(*Channel_41*)
	aPage_Channel[41].PARAM_NAME := 'Channel_41';
	aPage_Channel[41].PARAM_00   := 9;
	aPage_Channel[41].PARAM_01   := 1;
	aPage_Channel[41].PARAM_02   := 1;
	aPage_Channel[41].PARAM_03   := 1;
	aPage_Channel[41].PARAM_04   := 1;
	aPage_Channel[41].PARAM_05   := 1;
	aPage_Channel[41].PARAM_06   := 0;
	aPage_Channel[41].PARAM_07   := 0;
	aPage_Channel[41].PARAM_08   := 0;
	aPage_Channel[41].PARAM_09   := 0;
	aPage_Channel[41].PARAM_10   := 0;

(*Channel_42*)
	aPage_Channel[42].PARAM_NAME := 'Channel_42';
	aPage_Channel[42].PARAM_00   := 9;
	aPage_Channel[42].PARAM_01   := 1;
	aPage_Channel[42].PARAM_02   := 1;
	aPage_Channel[42].PARAM_03   := 1;
	aPage_Channel[42].PARAM_04   := 1;
	aPage_Channel[42].PARAM_05   := 1;
	aPage_Channel[42].PARAM_06   := 0;
	aPage_Channel[42].PARAM_07   := 0;
	aPage_Channel[42].PARAM_08   := 0;
	aPage_Channel[42].PARAM_09   := 0;
	aPage_Channel[42].PARAM_10   := 0;

(*Channel_43*)
	aPage_Channel[43].PARAM_NAME := 'Channel_43';
	aPage_Channel[43].PARAM_00   := 9;
	aPage_Channel[43].PARAM_01   := 1;
	aPage_Channel[43].PARAM_02   := 1;
	aPage_Channel[43].PARAM_03   := 1;
	aPage_Channel[43].PARAM_04   := 1;
	aPage_Channel[43].PARAM_05   := 1;
	aPage_Channel[43].PARAM_06   := 0;
	aPage_Channel[43].PARAM_07   := 0;
	aPage_Channel[43].PARAM_08   := 0;
	aPage_Channel[43].PARAM_09   := 0;
	aPage_Channel[43].PARAM_10   := 0;

(*Channel_44*)
	aPage_Channel[44].PARAM_NAME := 'Channel_44';
	aPage_Channel[44].PARAM_00   := 9;
	aPage_Channel[44].PARAM_01   := 1;
	aPage_Channel[44].PARAM_02   := 1;
	aPage_Channel[44].PARAM_03   := 1;
	aPage_Channel[44].PARAM_04   := 1;
	aPage_Channel[44].PARAM_05   := 1;
	aPage_Channel[44].PARAM_06   := 0;
	aPage_Channel[44].PARAM_07   := 0;
	aPage_Channel[44].PARAM_08   := 0;
	aPage_Channel[44].PARAM_09   := 0;
	aPage_Channel[44].PARAM_10   := 0;

(*Channel_45*)
	aPage_Channel[45].PARAM_NAME := 'Channel_45';
	aPage_Channel[45].PARAM_00   := 9;
	aPage_Channel[45].PARAM_01   := 1;
	aPage_Channel[45].PARAM_02   := 1;
	aPage_Channel[45].PARAM_03   := 1;
	aPage_Channel[45].PARAM_04   := 1;
	aPage_Channel[45].PARAM_05   := 1;
	aPage_Channel[45].PARAM_06   := 0;
	aPage_Channel[45].PARAM_07   := 0;
	aPage_Channel[45].PARAM_08   := 0;
	aPage_Channel[45].PARAM_09   := 0;
	aPage_Channel[45].PARAM_10   := 0;

(*Channel_46*)
	aPage_Channel[46].PARAM_NAME := 'Channel_46';
	aPage_Channel[46].PARAM_00   := 9;
	aPage_Channel[46].PARAM_01   := 1;
	aPage_Channel[46].PARAM_02   := 1;
	aPage_Channel[46].PARAM_03   := 1;
	aPage_Channel[46].PARAM_04   := 1;
	aPage_Channel[46].PARAM_05   := 1;
	aPage_Channel[46].PARAM_06   := 0;
	aPage_Channel[46].PARAM_07   := 0;
	aPage_Channel[46].PARAM_08   := 0;
	aPage_Channel[46].PARAM_09   := 0;
	aPage_Channel[46].PARAM_10   := 0;

(*Channel_47*)
	aPage_Channel[47].PARAM_NAME := 'Channel_47';
	aPage_Channel[47].PARAM_00   := 9;
	aPage_Channel[47].PARAM_01   := 1;
	aPage_Channel[47].PARAM_02   := 1;
	aPage_Channel[47].PARAM_03   := 1;
	aPage_Channel[47].PARAM_04   := 1;
	aPage_Channel[47].PARAM_05   := 1;
	aPage_Channel[47].PARAM_06   := 0;
	aPage_Channel[47].PARAM_07   := 0;
	aPage_Channel[47].PARAM_08   := 0;
	aPage_Channel[47].PARAM_09   := 0;
	aPage_Channel[47].PARAM_10   := 0;

(*Channel_48*)
	aPage_Channel[48].PARAM_NAME := 'Channel_48';
	aPage_Channel[48].PARAM_00   := 9;
	aPage_Channel[48].PARAM_01   := 1;
	aPage_Channel[48].PARAM_02   := 1;
	aPage_Channel[48].PARAM_03   := 1;
	aPage_Channel[48].PARAM_04   := 1;
	aPage_Channel[48].PARAM_05   := 1;
	aPage_Channel[48].PARAM_06   := 0;
	aPage_Channel[48].PARAM_07   := 0;
	aPage_Channel[48].PARAM_08   := 0;
	aPage_Channel[48].PARAM_09   := 0;
	aPage_Channel[48].PARAM_10   := 0;

(*Channel_49*)
	aPage_Channel[49].PARAM_NAME := 'Channel_49';
	aPage_Channel[49].PARAM_00   := 9;
	aPage_Channel[49].PARAM_01   := 1;
	aPage_Channel[49].PARAM_02   := 1;
	aPage_Channel[49].PARAM_03   := 1;
	aPage_Channel[49].PARAM_04   := 1;
	aPage_Channel[49].PARAM_05   := 1;
	aPage_Channel[49].PARAM_06   := 0;
	aPage_Channel[49].PARAM_07   := 0;
	aPage_Channel[49].PARAM_08   := 0;
	aPage_Channel[49].PARAM_09   := 0;
	aPage_Channel[49].PARAM_10   := 0;

(*Channel_50*)
	aPage_Channel[50].PARAM_NAME := 'Channel_50';
	aPage_Channel[50].PARAM_00   := 9;
	aPage_Channel[50].PARAM_01   := 1;
	aPage_Channel[50].PARAM_02   := 1;
	aPage_Channel[50].PARAM_03   := 1;
	aPage_Channel[50].PARAM_04   := 1;
	aPage_Channel[50].PARAM_05   := 1;
	aPage_Channel[50].PARAM_06   := 0;
	aPage_Channel[50].PARAM_07   := 0;
	aPage_Channel[50].PARAM_08   := 0;
	aPage_Channel[50].PARAM_09   := 0;
	aPage_Channel[50].PARAM_10   := 0;

(*Channel_51*)
	aPage_Channel[51].PARAM_NAME := 'Channel_51';
	aPage_Channel[51].PARAM_00   := 9;
	aPage_Channel[51].PARAM_01   := 1;
	aPage_Channel[51].PARAM_02   := 1;
	aPage_Channel[51].PARAM_03   := 1;
	aPage_Channel[51].PARAM_04   := 1;
	aPage_Channel[51].PARAM_05   := 1;
	aPage_Channel[51].PARAM_06   := 0;
	aPage_Channel[51].PARAM_07   := 0;
	aPage_Channel[51].PARAM_08   := 0;
	aPage_Channel[51].PARAM_09   := 0;
	aPage_Channel[51].PARAM_10   := 0;

(*Channel_52*)
	aPage_Channel[52].PARAM_NAME := 'Channel_52';
	aPage_Channel[52].PARAM_00   := 9;
	aPage_Channel[52].PARAM_01   := 1;
	aPage_Channel[52].PARAM_02   := 1;
	aPage_Channel[52].PARAM_03   := 1;
	aPage_Channel[52].PARAM_04   := 1;
	aPage_Channel[52].PARAM_05   := 1;
	aPage_Channel[52].PARAM_06   := 0;
	aPage_Channel[52].PARAM_07   := 0;
	aPage_Channel[52].PARAM_08   := 0;
	aPage_Channel[52].PARAM_09   := 0;
	aPage_Channel[52].PARAM_10   := 0;

(*Channel_53*)
	aPage_Channel[53].PARAM_NAME := 'Channel_53';
	aPage_Channel[53].PARAM_00   := 9;
	aPage_Channel[53].PARAM_01   := 1;
	aPage_Channel[53].PARAM_02   := 1;
	aPage_Channel[53].PARAM_03   := 1;
	aPage_Channel[53].PARAM_04   := 1;
	aPage_Channel[53].PARAM_05   := 1;
	aPage_Channel[53].PARAM_06   := 0;
	aPage_Channel[53].PARAM_07   := 0;
	aPage_Channel[53].PARAM_08   := 0;
	aPage_Channel[53].PARAM_09   := 0;
	aPage_Channel[53].PARAM_10   := 0;

(*Channel_54*)
	aPage_Channel[54].PARAM_NAME := 'Channel_54';
	aPage_Channel[54].PARAM_00   := 9;
	aPage_Channel[54].PARAM_01   := 1;
	aPage_Channel[54].PARAM_02   := 1;
	aPage_Channel[54].PARAM_03   := 1;
	aPage_Channel[54].PARAM_04   := 1;
	aPage_Channel[54].PARAM_05   := 1;
	aPage_Channel[54].PARAM_06   := 0;
	aPage_Channel[54].PARAM_07   := 0;
	aPage_Channel[54].PARAM_08   := 0;
	aPage_Channel[54].PARAM_09   := 0;
	aPage_Channel[54].PARAM_10   := 0;

(*Channel_55*)
	aPage_Channel[55].PARAM_NAME := 'Channel_55';
	aPage_Channel[55].PARAM_00   := 9;
	aPage_Channel[55].PARAM_01   := 1;
	aPage_Channel[55].PARAM_02   := 1;
	aPage_Channel[55].PARAM_03   := 1;
	aPage_Channel[55].PARAM_04   := 1;
	aPage_Channel[55].PARAM_05   := 1;
	aPage_Channel[55].PARAM_06   := 0;
	aPage_Channel[55].PARAM_07   := 0;
	aPage_Channel[55].PARAM_08   := 0;
	aPage_Channel[55].PARAM_09   := 0;
	aPage_Channel[55].PARAM_10   := 0;

(*Channel_56*)
	aPage_Channel[56].PARAM_NAME := 'Channel_56';
	aPage_Channel[56].PARAM_00   := 9;
	aPage_Channel[56].PARAM_01   := 1;
	aPage_Channel[56].PARAM_02   := 1;
	aPage_Channel[56].PARAM_03   := 1;
	aPage_Channel[56].PARAM_04   := 1;
	aPage_Channel[56].PARAM_05   := 1;
	aPage_Channel[56].PARAM_06   := 0;
	aPage_Channel[56].PARAM_07   := 0;
	aPage_Channel[56].PARAM_08   := 0;
	aPage_Channel[56].PARAM_09   := 0;
	aPage_Channel[56].PARAM_10   := 0;

(*Channel_57*)
	aPage_Channel[57].PARAM_NAME := 'Channel_57';
	aPage_Channel[57].PARAM_00   := 9;
	aPage_Channel[57].PARAM_01   := 1;
	aPage_Channel[57].PARAM_02   := 1;
	aPage_Channel[57].PARAM_03   := 1;
	aPage_Channel[57].PARAM_04   := 1;
	aPage_Channel[57].PARAM_05   := 1;
	aPage_Channel[57].PARAM_06   := 0;
	aPage_Channel[57].PARAM_07   := 0;
	aPage_Channel[57].PARAM_08   := 0;
	aPage_Channel[57].PARAM_09   := 0;
	aPage_Channel[57].PARAM_10   := 0;

(*Channel_58*)
	aPage_Channel[58].PARAM_NAME := 'Channel_58';
	aPage_Channel[58].PARAM_00   := 9;
	aPage_Channel[58].PARAM_01   := 1;
	aPage_Channel[58].PARAM_02   := 1;
	aPage_Channel[58].PARAM_03   := 1;
	aPage_Channel[58].PARAM_04   := 1;
	aPage_Channel[58].PARAM_05   := 1;
	aPage_Channel[58].PARAM_06   := 0;
	aPage_Channel[58].PARAM_07   := 0;
	aPage_Channel[58].PARAM_08   := 0;
	aPage_Channel[58].PARAM_09   := 0;
	aPage_Channel[58].PARAM_10   := 0;

(*Channel_59*)
	aPage_Channel[59].PARAM_NAME := 'Channel_59';
	aPage_Channel[59].PARAM_00   := 9;
	aPage_Channel[59].PARAM_01   := 1;
	aPage_Channel[59].PARAM_02   := 1;
	aPage_Channel[59].PARAM_03   := 1;
	aPage_Channel[59].PARAM_04   := 1;
	aPage_Channel[59].PARAM_05   := 1;
	aPage_Channel[59].PARAM_06   := 0;
	aPage_Channel[59].PARAM_07   := 0;
	aPage_Channel[59].PARAM_08   := 0;
	aPage_Channel[59].PARAM_09   := 0;
	aPage_Channel[59].PARAM_10   := 0;

(*Channel_60*)
	aPage_Channel[60].PARAM_NAME := 'Channel_60';
	aPage_Channel[60].PARAM_00   := 9;
	aPage_Channel[60].PARAM_01   := 1;
	aPage_Channel[60].PARAM_02   := 1;
	aPage_Channel[60].PARAM_03   := 1;
	aPage_Channel[60].PARAM_04   := 1;
	aPage_Channel[60].PARAM_05   := 1;
	aPage_Channel[60].PARAM_06   := 0;
	aPage_Channel[60].PARAM_07   := 0;
	aPage_Channel[60].PARAM_08   := 0;
	aPage_Channel[60].PARAM_09   := 0;
	aPage_Channel[60].PARAM_10   := 0;

(*Channel_61*)
	aPage_Channel[61].PARAM_NAME := 'Channel_61';
	aPage_Channel[61].PARAM_00   := 9;
	aPage_Channel[61].PARAM_01   := 1;
	aPage_Channel[61].PARAM_02   := 1;
	aPage_Channel[61].PARAM_03   := 1;
	aPage_Channel[61].PARAM_04   := 1;
	aPage_Channel[61].PARAM_05   := 1;
	aPage_Channel[61].PARAM_06   := 0;
	aPage_Channel[61].PARAM_07   := 0;
	aPage_Channel[61].PARAM_08   := 0;
	aPage_Channel[61].PARAM_09   := 0;
	aPage_Channel[61].PARAM_10   := 0;

(*Channel_62*)
	aPage_Channel[62].PARAM_NAME := 'Channel_62';
	aPage_Channel[62].PARAM_00   := 9;
	aPage_Channel[62].PARAM_01   := 1;
	aPage_Channel[62].PARAM_02   := 1;
	aPage_Channel[62].PARAM_03   := 1;
	aPage_Channel[62].PARAM_04   := 1;
	aPage_Channel[62].PARAM_05   := 1;
	aPage_Channel[62].PARAM_06   := 0;
	aPage_Channel[62].PARAM_07   := 0;
	aPage_Channel[62].PARAM_08   := 0;
	aPage_Channel[62].PARAM_09   := 0;
	aPage_Channel[62].PARAM_10   := 0;

(*Channel_63*)
	aPage_Channel[63].PARAM_NAME := 'Channel_63';
	aPage_Channel[63].PARAM_00   := 9;
	aPage_Channel[63].PARAM_01   := 1;
	aPage_Channel[63].PARAM_02   := 1;
	aPage_Channel[63].PARAM_03   := 1;
	aPage_Channel[63].PARAM_04   := 1;
	aPage_Channel[63].PARAM_05   := 1;
	aPage_Channel[63].PARAM_06   := 0;
	aPage_Channel[63].PARAM_07   := 0;
	aPage_Channel[63].PARAM_08   := 0;
	aPage_Channel[63].PARAM_09   := 0;
	aPage_Channel[63].PARAM_10   := 0;

(*-----------------------------------------------------------------------------------------------------------------------------------------------------------------------------------*)
(**)

	DefaultSettingsUnitModeRecovery;

	bCurrModeChange := 0;

END_IF;
END_PROGRAM

(* POU Default_Settings/Parameter_Recovery_processing, ST *)
PROGRAM Parameter_Recovery_processing

VAR_INPUT
	bInit        : BOOL;
END_VAR

VAR
	instFRAMRead : FRAMREAD;
	i            : INT;
END_VAR
(*-----------------------------------------------------------------------------------------------------------------------------------------------------------------------------------*)
(*Извлечение из энергонезависимой памяти установочных параметров, коэффициентов и формирование массивов, соответствующих измерительным каналам*)

    instFRAMRead(Enable := 1, SRC := iMemAdrCurrMode,                LEN := 4,  DST := ADR(dwCurrMode));(*Читаем идентификатор режима*)
    instFRAMRead(Enable := 1, SRC := iMemAdrCHANNEL_INDEX,           LEN := 4,  DST := ADR(dwCHANNEL_INDEX));(**)

    instFRAMRead(Enable := 1, SRC := iMemAdrSet_GN2TempManual,    LEN := 4, DST := ADR(rSet_GN2TempManual));
IF rSet_GN2TempManual > 50 THEN rSet_GN2TempManual := 50; END_IF;
IF rSet_GN2TempManual <  5 THEN rSet_GN2TempManual :=  5; END_IF;

    instFRAMRead(Enable := 1, SRC := iMemAdrSet_GN2OverPres,      LEN := 4, DST := ADR(rSet_GN2OverPres));
    instFRAMRead(Enable := 1, SRC := iMemAdrSet_BoostPresManual,  LEN := 4, DST := ADR(rSet_BoostPresManual));

    instFRAMRead(Enable := 1, SRC := iMemAdrSet_GN2Rate,          LEN := 4, DST := ADR(rSet_GN2Rate));
IF rSet_GN2Rate > 85 THEN rSet_GN2Rate := 85; END_IF;

    instFRAMRead(Enable := 1, SRC := iMemAdrSet_LN2SaturTemp,     LEN := 4, DST := ADR(rSet_LN2SaturTemp));

FOR i := 0 TO 63 DO
	instFRAMRead(Enable := 1, SRC := iMemAdrArrayParamName + i * 32, LEN := 32, DST := ADR(aPage_Channel[i].PARAM_NAME));

	instFRAMRead(Enable := 1, SRC := iMemAdrArrayParam00 + i * 4,    LEN := 4,  DST := ADR(aPage_Channel[i].PARAM_00));
	instFRAMRead(Enable := 1, SRC := iMemAdrArrayParam01 + i * 4,    LEN := 4,  DST := ADR(aPage_Channel[i].PARAM_01));
	instFRAMRead(Enable := 1, SRC := iMemAdrArrayParam02 + i * 4,    LEN := 4,  DST := ADR(aPage_Channel[i].PARAM_02));
	instFRAMRead(Enable := 1, SRC := iMemAdrArrayParam03 + i * 4,    LEN := 4,  DST := ADR(aPage_Channel[i].PARAM_03));
	instFRAMRead(Enable := 1, SRC := iMemAdrArrayParam04 + i * 4,    LEN := 4,  DST := ADR(aPage_Channel[i].PARAM_04));
	instFRAMRead(Enable := 1, SRC := iMemAdrArrayParam05 + i * 4,    LEN := 4,  DST := ADR(aPage_Channel[i].PARAM_05));
	instFRAMRead(Enable := 1, SRC := iMemAdrArrayParam06 + i * 4,    LEN := 4,  DST := ADR(aPage_Channel[i].PARAM_06));
	instFRAMRead(Enable := 1, SRC := iMemAdrArrayParam07 + i * 4,    LEN := 4,  DST := ADR(aPage_Channel[i].PARAM_07));

	instFRAMRead(Enable := 1, SRC := iMemAdrArrayParam09 + i * 4,    LEN := 4,  DST := ADR(aPage_Channel[i].PARAM_09));
	instFRAMRead(Enable := 1, SRC := iMemAdrArrayParam10 + i * 4,    LEN := 4,  DST := ADR(aPage_Channel[i].PARAM_10));

(*Накладываем ограничения на извлекаемые из памяти коэффициенты для аналоговых каналов*)
	IF aPage_Channel[i].PARAM_00 = 0 THEN
		IF aPage_Channel[i].PARAM_05 < 10   THEN aPage_Channel[i].PARAM_05 := 10;   END_IF;
		IF aPage_Channel[i].PARAM_05 > 2_000 THEN aPage_Channel[i].PARAM_05 := 2_000; END_IF;
	END_IF;

(*Накладываем ограничения на извлекаемые из памяти коэффициенты для частотных каналов*)
	IF aPage_Channel[i].PARAM_00 = 1 THEN
		aPage_Channel[i].PARAM_05 := 1_000;
	END_IF;

(*Накладываем ограничения на извлекаемые из памяти коэффициенты для каналов ШИМ*)
	IF aPage_Channel[i].PARAM_00 = 2 THEN
		IF aPage_Channel[i].PARAM_05 < 200   THEN aPage_Channel[i].PARAM_05 := 200;   END_IF;
		IF aPage_Channel[i].PARAM_05 > 32_767 THEN aPage_Channel[i].PARAM_05 := 32_767; END_IF;
	END_IF;

END_FOR;
END_PROGRAM

(* POU AIN_RAW_processing, ST *)
PROGRAM AIN_RAW_processing

VAR_INPUT
	bInit      : BOOL;
END_VAR

VAR
	i          : INT := 0;

	iCycleZero : INT := 0;
	t          : INT := 0;
END_VAR
(*-----------------------------------------------------------------------------------------------------------------------------------------------------------------------------------*)
(*Снимаем текущие значения аналоговых каналов*)

(*Массив исходных значений в REAL*)
rArrayDataRAWADC[ 1] := WORD_TO_REAL(%IW3);(*1-08*)
rArrayDataRAWADC[ 2] := WORD_TO_REAL(%IW4);(*1-27*)
rArrayDataRAWADC[ 3] := WORD_TO_REAL(%IW5);(*1-09*)
rArrayDataRAWADC[ 4] := WORD_TO_REAL(%IW6);(*1-28*)
rArrayDataRAWADC[ 5] := WORD_TO_REAL(%IW7);(*1-10*)
rArrayDataRAWADC[ 6] := WORD_TO_REAL(%IW8);(*1-29*)
rArrayDataRAWADC[ 7] := WORD_TO_REAL(%IW9);(*1-11*)
rArrayDataRAWADC[ 8] := WORD_TO_REAL(%IW10);(*1-30*)

rArrayDataRAWADC[ 9] := 0;(*2-08*)
rArrayDataRAWADC[10] := 0;(*2-27*)
rArrayDataRAWADC[11] := 0;(*2-09*)
rArrayDataRAWADC[12] := 0;(*2-28*)
rArrayDataRAWADC[13] := 0;(*2-10*)
rArrayDataRAWADC[14] := 0;(*2-29*)
rArrayDataRAWADC[15] := 0;(*2-11*)
rArrayDataRAWADC[16] := 0;(*2-30*)

(*-----------------------------------------------------------------------------------------------------------------------------------------------------------------------------------*)
(**)

IF bInit = 1 THEN iCycleZero := 10; END_IF;

IF iCycleZero > 0 THEN
	FOR t := 1 TO 16 DO
		rArrayDataRAWADC[t] := 0;
	END_FOR;
	bResetErrors := 1;
	iCycleZero := iCycleZero - 1;
END_IF;

(*-----------------------------------------------------------------------------------------------------------------------------------------------------------------------------------*)
(*Обработка обрывов (значение меньше минимально допустимого) и КЗ (значение больше максимально допустимого) по входу канала*)

FOR i := 1 TO 16 DO

	IF rArrayDataRAWADC[i] > rADC_ValueHigh
		THEN bArrayErrorADC[i * 2 - 1] := 1;(**)
		ELSE bArrayErrorADC[i * 2 - 1] := 0;(**)
	END_IF;

	IF rArrayDataRAWADC[i] < rADC_ValueLow (**)
		THEN bArrayErrorADC[i * 2] := 1;(**)
		ELSE bArrayErrorADC[i * 2] := 0;(**)
	END_IF;

END_FOR;

(*-----------------------------------------------------------------------------------------------------------------------------------------------------------------------------------*)
(*Подготовка для выдачи в CAN обрывов и коротких замыканий по входам АЦП*)

dwErrorADC_MS.0  := bArrayErrorADC[ 1];
dwErrorADC_MS.1  := bArrayErrorADC[ 2];
dwErrorADC_MS.2  := bArrayErrorADC[ 3];
dwErrorADC_MS.3  := bArrayErrorADC[ 4];
dwErrorADC_MS.4  := bArrayErrorADC[ 5];
dwErrorADC_MS.5  := bArrayErrorADC[ 6];
dwErrorADC_MS.6  := bArrayErrorADC[ 7];
dwErrorADC_MS.7  := bArrayErrorADC[ 8];

dwErrorADC_MS.8  := bArrayErrorADC[ 9];
dwErrorADC_MS.9  := bArrayErrorADC[10];
dwErrorADC_MS.10 := bArrayErrorADC[11];
dwErrorADC_MS.11 := bArrayErrorADC[12];
dwErrorADC_MS.12 := bArrayErrorADC[13];
dwErrorADC_MS.13 := bArrayErrorADC[14];
dwErrorADC_MS.14 := bArrayErrorADC[15];
dwErrorADC_MS.15 := bArrayErrorADC[16];

dwErrorADC_MS.16 := bArrayErrorADC[17];
dwErrorADC_MS.17 := bArrayErrorADC[18];
dwErrorADC_MS.18 := bArrayErrorADC[19];
dwErrorADC_MS.19 := bArrayErrorADC[20];
dwErrorADC_MS.20 := bArrayErrorADC[21];
dwErrorADC_MS.21 := bArrayErrorADC[22];
dwErrorADC_MS.22 := bArrayErrorADC[23];
dwErrorADC_MS.23 := bArrayErrorADC[24];

dwErrorADC_MS.24 := bArrayErrorADC[25];
dwErrorADC_MS.25 := bArrayErrorADC[26];
dwErrorADC_MS.26 := bArrayErrorADC[27];
dwErrorADC_MS.27 := bArrayErrorADC[28];
dwErrorADC_MS.28 := bArrayErrorADC[29];
dwErrorADC_MS.29 := bArrayErrorADC[30];
dwErrorADC_MS.30 := bArrayErrorADC[31];
dwErrorADC_MS.31 := bArrayErrorADC[32];

(*-----------------------------------------------------------------------------------------------------------------------------------------------------------------------------------*)
(**)

dwErrorADC_SL1 := 16#FFFF;

(*-----------------------------------------------------------------------------------------------------------------------------------------------------------------------------------*)
(**)

dwErrorADC_SL2 := 16#FFFF;


(*-----------------------------------------------------------------------------------------------------------------------------------------------------------------------------------*)
(**)

dwErrorADC_SL3 := 16#FFFF;
END_PROGRAM

(* POU PIN_RAW_processing, ST *)
PROGRAM PIN_RAW_processing

VAR_INPUT
	bInit          : BOOL;
END_VAR

VAR
	Freq_0         : FREQUENCY;
	Freq_1         : FREQUENCY;
	Freq_2         : FREQUENCY;
	Freq_3         : FREQUENCY;

	Period_0       : PERIOD;
	Period_1       : PERIOD;
	Period_2       : PERIOD;
	Period_3       : PERIOD;

	rFreqIn_0      : REAL;(*Частотный канал 0, контроллер #1*)
	rFreqIn_1      : REAL;(*Частотный канал 1, контроллер #1*)
	rFreqIn_2      : REAL;(*Частотный канал 2, контроллер #1*)
	rFreqIn_3      : REAL;(*Частотный канал 3, контроллер #1*)

	dwPeriodIn_0   : DWORD;(*Канал измерения периода 0, контроллер #1*)
	dwPeriodIn_1   : DWORD;(*Канал измерения периода 1, контроллер #1*)
	dwPeriodIn_2   : DWORD;(*Канал измерения периода 2, контроллер #1*)
	dwPeriodIn_3   : DWORD;(*Канал измерения периода 3, контроллер #1*)

	rFreqPerIn_0   : REAL;(*Канал измерения периода 0, контроллер #1*)
	rFreqPerIn_1   : REAL;(*Канал измерения периода 1, контроллер #1*)
	rFreqPerIn_2   : REAL;(*Канал измерения периода 2, контроллер #1*)
	rFreqPerIn_3   : REAL;(*Канал измерения периода 3, контроллер #1*)

	tElapsedTime_0 : TIME;(*Канал измерения периода 0, контроллер #1*)
	tElapsedTime_1 : TIME;(*Канал измерения периода 1, контроллер #1*)
	tElapsedTime_2 : TIME;(*Канал измерения периода 2, контроллер #1*)
	tElapsedTime_3 : TIME;(*Канал измерения периода 3, контроллер #1*)

	TimeOff                 : TP;
	bTimeOff                : BOOL;
	diCurrentEngineRPM_Prev : DINT;
END_VAR
(*-----------------------------------------------------------------------------------------------------------------------------------------------------------------------------------*)
(*Снимаем текущие значения частотных каналов*)

Freq_0(Init := bInit, Channel := 0, TimeBase := T#1000ms, F => rFreqIn_0);
Freq_1(Init := bInit, Channel := 1, TimeBase := T#1000ms, F => rFreqIn_1);
Freq_2(Init := bInit, Channel := 2, TimeBase := T#1000ms, F => rFreqIn_2);
Freq_3(Init := bInit, Channel := 3, TimeBase := T#1000ms, F => rFreqIn_3);

(*-----------------------------------------------------------------------------------------------------------------------------------------------------------------------------------*)
(*Снимаем текущие значения каналов измерения периода*)

Period_0(Init := bInit, Channel := 0, Periods := 82, C => dwPeriodIn_0, F => rFreqPerIn_0, ET => tElapsedTime_0);
Period_1(Init := bInit, Channel := 1, Periods := 82, C => dwPeriodIn_1, F => rFreqPerIn_1, ET => tElapsedTime_1);
Period_2(Init := bInit, Channel := 2, Periods := 82, C => dwPeriodIn_2, F => rFreqPerIn_2, ET => tElapsedTime_2);
Period_3(Init := bInit, Channel := 3, Periods := 82, C => dwPeriodIn_3, F => rFreqPerIn_3, ET => tElapsedTime_3);

(*-----------------------------------------------------------------------------------------------------------------------------------------------------------------------------------*)
(*Собираем текущие значения частотных каналов в массив*)
(*Если частота больше 950 Гц, то используем частотные каналы*)
(*Если частота меньше 950 Гц, то используем каналы измерения периода*)

IF rFreqIn_0 > 950
THEN
	rArrayDataRAWPIN[1] := rFreqIn_0;
ELSE
	rArrayDataRAWPIN[1] := rFreqPerIn_0;
END_IF;

IF rFreqIn_1 > 950
THEN
	rArrayDataRAWPIN[2] := rFreqIn_1;
ELSE
	rArrayDataRAWPIN[2] := rFreqPerIn_1;
END_IF;

IF rFreqIn_2 > 950
THEN
	rArrayDataRAWPIN[3] := rFreqIn_2;
ELSE
	rArrayDataRAWPIN[3] := rFreqPerIn_2;
END_IF;

IF rFreqIn_3 > 950
THEN
	rArrayDataRAWPIN[4] := rFreqIn_3;
ELSE
	rArrayDataRAWPIN[4] := rFreqPerIn_3;
END_IF;

(*-----------------------------------------------------------------------------------------------------------------------------------------------------------------------------------*)
(**)

TimeOff(IN := , PT := T#5S, Q => , ET => );

IF diCurrentEngineRPM_Prev < 500 AND diCurrentEngineRPM > 500
THEN
	TimeOff.IN := 1;
END_IF;

IF TimeOff.Q = 1
THEN
	rArrayDataRAWPIN[1] := 0;
	rArrayDataRAWPIN[2] := 0;
	rArrayDataRAWPIN[3] := 0;
	rArrayDataRAWPIN[4] := 0;
	TimeOff.IN := 0;
END_IF;

IF diCurrentEngineRPM < 600
THEN
	rArrayDataRAWPIN[1] := 0;
	rArrayDataRAWPIN[2] := 0;
	rArrayDataRAWPIN[3] := 0;
	rArrayDataRAWPIN[4] := 0;
END_IF;

diCurrentEngineRPM_Prev := diCurrentEngineRPM;

(*-----------------------------------------------------------------------------------------------------------------------------------------------------------------------------------*)
(**)

rArrayDataRAWPIN[5] := 0;
rArrayDataRAWPIN[6] := 0;
rArrayDataRAWPIN[7] := 0;
rArrayDataRAWPIN[8] := 0;

(*-----------------------------------------------------------------------------------------------------------------------------------------------------------------------------------*)
(**)
END_PROGRAM

(* POU DIN_processing, ST *)
PROGRAM DIN_processing

VAR_INPUT
	bInit : BOOL;
END_VAR

VAR
END_VAR
(*-----------------------------------------------------------------------------------------------------------------------------------------------------------------------------------*)
(**)

dwInputState := 16#0000;

bIX_TriplexRPMAutoMode   := %IX1.8;  (*1-39*)
bIX_HydHeatPresAutoMode  := %IX1.9;  (*1-03*)
bIX_BoostPresAutoMode    := %IX1.10; (*1-40*)
bIX_BlockOff             := %IX1.15; (*1-04*)
bIX_EngineStopped        := %IX2.1;  (*1-49*)
IX_Test                  := %IX2.3; (*1-50*)

dwInputState.0  := bIX_TriplexRPMAutoMode;
dwInputState.1  := bIX_HydHeatPresAutoMode;
dwInputState.2  := bIX_BoostPresAutoMode;
dwInputState.3  := 0;
dwInputState.4  := 0;
dwInputState.5  := bIX_BlockOff;
dwInputState.6  := bIX_EngineStopped;

dwInputState.11 := IX_Test;
END_PROGRAM

(* POU Steps/StepSet_processing, ST *)
PROGRAM StepSet_processing

VAR_INPUT
	bFirstIn : BOOL;(*Первый вход в программу*)
END_VAR

VAR
	byStep   : BYTE := 0;
	t        : INT  := 0;
	i: INT;
END_VAR
(*-----------------------------------------------------------------------------------------------------------------------------------------------------------------------------------*)
(*Сброс счетчика и флагов шагов в исходное состояние*)

IF  bFirstIn = TRUE THEN
	FOR byStep:=1 TO 5 DO bControlExecutionSteps[byStep] := FALSE; END_FOR;
	byRequestNextStep := 0;
	byCurrStep        := 0;
	byCurrentSubStep  := 0;
	byErrorStepPC     := 0;
	byErrorStepPan    := 0;
(*Ожиданиe разрешения начать выполнение по шагам*)
	W_REQ_STAGE       := 0;
	R_REQ_STAGE       := 0;
	RETURN;
END_IF;(* end IF  in_init ....*)

(*-----------------------------------------------------------------------------------------------------------------------------------------------------------------------------------*)
(*Установка шага: диапазон задаваемых оператором или программно (по условию) шагов от 1 до 5*)

byStep := 1;

WHILE (bControlExecutionSteps[byStep] AND byStep <= 5) DO

byStep := byStep + 1;

END_WHILE;

(*	IF ReceiveCAN.REQ_STAGE <> TransmitCAN.REQ_STAGE THEN (*запрос на следующий шаг от РС*)
		byRequestNextStep:=ReceiveCAN.REQ_STAGE;
	END_IF;
*)

IF byRequestNextStep = byStep THEN (*Если запрашиваемый шаг допустим, устанавливаем его*)
	byCurrStep := byRequestNextStep;
END_IF;

IF t >= 2 THEN (*В этом цикле задаем номер шага для автоматического прохождения*)
	t := 0;
	IF byRequestNextStep <= 5 THEN
		byRequestNextStep := byRequestNextStep + 1;
	ELSE
		byRequestNextStep := 0;
	END_IF;
ELSE
	t := t + 1;
END_IF;

FOR i := 1 TO 1000 DO
;
END_FOR;
END_PROGRAM

(* POU Steps/Step_0, ST *)
PROGRAM Step_0

VAR_INPUT
	wStepIn  : WORD;
END_VAR

VAR
	bFirstIn : BOOL;
END_VAR
(*-----------------------------------------------------------------------------------------------------------------------------------------------------------------------------------*)
(*Режим 0*)

IF wStepIn <> 0 THEN bFirstIn := TRUE; RETURN; END_IF;

(*-----------------------------------------------------------------------------------------------------------------------------------------------------------------------------------*)
(*Выполняем однократные действия шага*)

IF bFirstIn = 1 THEN (*формируем команды*)

	bQX_HydHeatPresContrMode := 0; (*Выключаем *)

	bStart                   := 0;

END_IF;

(*-----------------------------------------------------------------------------------------------------------------------------------------------------------------------------------*)
(*Выполняем циклические действия шага*)

(*bQX_EngineStarterBlock       := 1; (*Запуск двигателя заблокирован*)*)

(*-----------------------------------------------------------------------------------------------------------------------------------------------------------------------------------*)
(*Формируем разрешение перехода к следующему шагу*)

bControlExecutionSteps[wStepIn] := TRUE;
byStageCondition := 3;(*Окончен*)
END_PROGRAM

(* POU Steps/Step_1_Initialization, ST *)
PROGRAM Step_1_Initialization

VAR_INPUT
	wStepIn  : WORD;
END_VAR

VAR
	bFirstIn : BOOL;

	instFRAMWrite      : FRAMWRITE;
	instMemCpy         : MEMCPY;
	rStartLN2SaturTemp : REAL := -170;
END_VAR
(*-----------------------------------------------------------------------------------------------------------------------------------------------------------------------------------*)
(*Режим инициализации*)

IF wStepIn <> 1 THEN bFirstIn := 1; RETURN; END_IF;
IF NOT bControlExecutionSteps[wStepIn] THEN

(*-----------------------------------------------------------------------------------------------------------------------------------------------------------------------------------*)
(*Выполняем однократные действия шага*)

	IF bFirstIn = 1 THEN (*формируем команды*)

		bQX_HydHeatPresContrMode := 0; (*Выключаем *)

		bStart                   := 0;

		instFRAMWrite(Enable := 1, DST := iMemAdrSet_LN2SaturTemp, LEN := 4, SRC := ADR(rStartLN2SaturTemp));

		byStageCondition := 0;(*Работает*)
		bFirstIn := 0;
	END_IF;

(*-----------------------------------------------------------------------------------------------------------------------------------------------------------------------------------*)
(*Выполняем циклические действия шага*)

	(*bQX_EngineStarterBlock   := 1; (*Запуск двигателя заблокирован*)*)

(*-----------------------------------------------------------------------------------------------------------------------------------------------------------------------------------*)
(*Контроль  условий выполнения шага*)

	dwErrorConditionRunStep := 0;

(*Здесь должны быть условия*)

(*-----------------------------------------------------------------------------------------------------------------------------------------------------------------------------------*)
(*Формируем разрешение перехода к следующему шагу*)

	IF dwErrorConditionRunStep = 0 THEN
		bControlExecutionSteps[wStepIn] := 1;
		byStageCondition := 3;(*Окончен*)
	ELSE
		byStageCondition := 2;(*Работает с ошибкой*)
	END_IF;
END_IF;
END_PROGRAM

(* POU Steps/Step_2_Waiting, ST *)
PROGRAM Step_2_Waiting

VAR_INPUT
	wStepIn  : WORD;
END_VAR

VAR
	bFirstIn : BOOL;
END_VAR
(*-----------------------------------------------------------------------------------------------------------------------------------------------------------------------------------*)
(*Режим ожидания*)

IF wStepIn <> 2 THEN bFirstIn := TRUE; RETURN; END_IF;
IF NOT bControlExecutionSteps[wStepIn] THEN

(*-----------------------------------------------------------------------------------------------------------------------------------------------------------------------------------*)
(*Выполняем однократные действия шага*)

	IF bFirstIn = 1 THEN (*формируем команды*)
		bQX_HydHeatPresContrMode := 0; (*Выключаем *)
		bStart                   := 1;

		byStageCondition         := 0; (*Работает*)
		bFirstIn                 := 0;
	END_IF;

(*-----------------------------------------------------------------------------------------------------------------------------------------------------------------------------------*)
(*Выполняем циклические действия шага*)

	bQX_EngineStarterBlock       := 0; (*Разблокируем запуск двигателя. Если хотя бы один тумблер в "Авто", то в Error_processing запуск двигателя будет заблокирован*)

(*-----------------------------------------------------------------------------------------------------------------------------------------------------------------------------------*)
(*Контроль условий выполнения шага*)

	dwErrorConditionRunStep := 0;

	IF bStart <> 1 THEN dwErrorConditionRunStep := 1; END_IF; (*Работаем, пока не поступит команда "Старт"*)
	IF diCurrentEngineRPM < 100 THEN dwErrorConditionRunStep := dwErrorConditionRunStep OR 4; END_IF; (*Работаем, пока двигатель не начал вращаться*)
	IF (bIX_TriplexRPMAutoMode = 1 OR bIX_HydHeatPresAutoMode = 1 OR bIX_BoostPresAutoMode = 1) THEN dwErrorConditionRunStep := dwErrorConditionRunStep OR 8; END_IF; (*Работаем, пока хотя бы один тумблер в положении "Авто"*)

(*-----------------------------------------------------------------------------------------------------------------------------------------------------------------------------------*)
(*Формируем разрешение перехода к следующему шагу*)

	IF dwErrorConditionRunStep = 0 THEN
		bControlExecutionSteps[wStepIn] := TRUE;
		byStageCondition := 3;(*Окончен*)
	ELSE
		byStageCondition := 2;(*Работает с ошибкой*)
	END_IF;
END_IF;
END_PROGRAM

(* POU Steps/Step_3_Working, ST *)
PROGRAM Step_3_Working

VAR_INPUT
	wStepIn  : WORD;
END_VAR

VAR
	bFirstIn : BOOL;
END_VAR
(*-----------------------------------------------------------------------------------------------------------------------------------------------------------------------------------*)
(*Режим работы*)

IF wStepIn <> 3 THEN bFirstIn := TRUE; RETURN; END_IF;
IF NOT bControlExecutionSteps[wStepIn] THEN

(*-----------------------------------------------------------------------------------------------------------------------------------------------------------------------------------*)
(*Выполняем однократные действия шага*)

	IF bFirstIn = 1 THEN (*формируем команды*)

        bResetErrors := 1; (*Сбрасываем флаги сообщений об ошибках*)
		bQX_HydHeatPresContrMode := 0; (*Выключаем *)

		byStageCondition := 0;(*Работает*)
		bFirstIn := 0;
	END_IF;

(*-----------------------------------------------------------------------------------------------------------------------------------------------------------------------------------*)
(*Выполняем циклические действия шага*)

	bQX_EngineStarterBlock       := 0; (*Разблокируем запуск двигателя*)

(*-----------------------------------------------------------------------------------------------------------------------------------------------------------------------------------*)
(*Контроль условий выполнения шага*)

	dwErrorConditionRunStep := 0;

	IF bStart <> 0 THEN dwErrorConditionRunStep := 1; END_IF; (*Работаем, пока не поступит команда стоп (сброс команды старт)*)

(*-----------------------------------------------------------------------------------------------------------------------------------------------------------------------------------*)
(*Формируем разрешение перехода к следующему шагу*)

	IF dwErrorConditionRunStep = 0 THEN
		bControlExecutionSteps[wStepIn] := TRUE;
		byStageCondition := 3;(*Окончен*)
	ELSE
		byStageCondition := 2;(*Работает с ошибкой*)
	END_IF;
END_IF;
END_PROGRAM

(* POU Steps/Step_4_Ending, ST *)
PROGRAM Step_4_Ending

VAR_INPUT
	wStepIn  : WORD;
END_VAR

VAR
	bFirstIn : BOOL;
	byStep   : BYTE;
END_VAR
(*-----------------------------------------------------------------------------------------------------------------------------------------------------------------------------------*)
(*Режим завершения работы*)

IF wStepIn <> 4 THEN (*bFirstIn := TRUE;*) RETURN; END_IF;

(*-----------------------------------------------------------------------------------------------------------------------------------------------------------------------------------*)
(*Выполняем однократные действия шага*)



(*-----------------------------------------------------------------------------------------------------------------------------------------------------------------------------------*)
(*Выполняем циклические действия шага*)

	bQX_HydHeatPresContrMode := 0; (*Выключаем *)
	bQX_EngineStarterBlock   := 0; (*Разблокируем запуск двигателя*)

(*-----------------------------------------------------------------------------------------------------------------------------------------------------------------------------------*)
(*Контроль условий выполнения шага*)

	dwErrorConditionRunStep := 0;

(*-----------------------------------------------------------------------------------------------------------------------------------------------------------------------------------*)
(*Формируем разрешение перехода к следующему шагу (для последнего шага)*)

IF dwErrorConditionRunStep = 0 THEN
	(*bTimerFanAttemt := FALSE*);
	byStep := 1;
		WHILE byStep <= 5 DO
			bControlExecutionSteps[byStep] := 0;
			byStep := byStep + 1;
		END_WHILE;
	byCurrStep := 0;
	byCurrentSubStep := 0;
	byStageCondition := 3;(*Окончен*)
ELSE
	byStageCondition := 0;(*Работает*)
END_IF;
END_PROGRAM

(* POU Output Modules/Boost_processing, ST *)
PROGRAM Boost_processing

VAR_INPUT
	bFirstIn                  : BOOL;
END_VAR

VAR
	bIX_BoostPresAutoModePrev : BOOL :=    0;
	bLN2_WorkOverTemp         : BOOL :=    0;

	(*bQX_BoostPresEmergStop    : BOOL :=    0;*)

	PID_3                     : PID;
 	PID_3_Reset               : BOOL :=    0;
	PID_3_Limits              : BOOL :=    0;
	PID_3_Manual              : BOOL :=    0;
	PID_3_Y_Manual            : REAL :=    0;
	PID_3_Y_Max               : REAL :=  400 (*1000*);
	PID_3_Overflow            : BOOL :=    0;

	instFRAMWrite             : FRAMWRITE;

(*Переменные для канала ШИМ*)
	PWM3                      : PWM1000;(*Выход ШИМ канал 2 на пин 46*)
	BoostPresFreqPWM          : FREQ_CHANGE_PWM;
    bBoostPresEnablePrev      : BOOL;

	TimerOn                   : TP;(*Задержка 5 секунд*)
	bTimerOnStart             : BOOL := 0;
	bTimerOnOut               : BOOL := 0;
	bFlagCycle                : BOOL := 0;
END_VAR
(*-----------------------------------------------------------------------------------------------------------------------------------------------------------------------------------*)
(*Управляем давлением нагнетания (подпитывающий насос)*)

TimerOn;
bTimerOnOut:=TimerOn.Q;

(*-----------------------------------------------------------------------------------------------------------------------------------------------------------------------------------*)
(*bErrorNumber17 - Ошибка 17. Центробеж. насос. Температура жидкого азота выше допустимого*)

IF byCurrStep = 3 AND bBoostPresDisparity = 1 AND rIW_LN2_Temp > rSet_LN2SaturTemp
THEN
	bErrorNumber17  := 1;(*РАБОТАЕМ С ПРЕДУПРЕЖДЕНИЕМ*)
	dwHornEnable.17 := 0;(*Сирена отключена*)
ELSE
	bErrorNumber17  := 0;
	dwHornEnable.17 := 0;
END_IF;

(*-----------------------------------------------------------------------------------------------------------------------------------------------------------------------------------*)
(*Возврат корректированного давления нагнетания после повторного возврата в режим "Авто"*)

IF bIX_BoostPresAutoModePrev = 0 AND bIX_BoostPresAutoMode = 1
THEN
	instFRAMWrite(Enable := 1, DST := iMemAdrSet_BoostPresManual, LEN := 4, SRC := ADR(rSet_BoostPresAuto));
	bLN2_WorkOverTemp := 0;
END_IF;

(*-----------------------------------------------------------------------------------------------------------------------------------------------------------------------------------*)
(*Формируем разрешение автоматического режима при положении тумблера "Авто"*)

IF byCurrStep = 3 AND bIX_BoostPresAutoMode = 1 (*AND bQX_BoostPresEmergStop = 1*) AND rIW_LN2_Temp <= rSet_LN2SaturTemp AND bLN2_WorkOverTemp = 0 AND bIX_BlockOff = 0 AND bCommomErrorADC = 0
THEN
	bBoostPresEnable := 1;
	IF bSet_BoostPresManual = 1
	THEN
		rSet_BoostPres := rSet_BoostPresManual;
	ELSE
		rSet_BoostPres := rSet_BoostPresAuto;
	END_IF;
	bQX_BoostPresContrMode := 1;(*Зеленой лампочкой светим постоянно*)
ELSE
	bBoostPresEnable := 0;
	bQX_BoostPresContrMode := 0;(*Зеленую лампочку погасили*)
END_IF;

(*-----------------------------------------------------------------------------------------------------------------------------------------------------------------------------------*)
(*Формируем признак отключенного автоматического режима при положении тумблера "Авто"*)

IF (*byCurrStep = 3 AND*) bIX_BoostPresAutoMode = 1 AND bBoostPresEnable = 0
THEN
	bBoostPresDisparity := 1;
	bQX_BoostPresContrMode := bTimerBlinkOut;(*Зеленой лампочкой мигаем*)
ELSE
	bBoostPresDisparity := 0;
END_IF;

(*-----------------------------------------------------------------------------------------------------------------------------------------------------------------------------------*)
(*bErrorNumber20 - Ошибка 20. Центробеж. насос. Давление подпитки ниже допустимого*)

IF bBoostPresEnablePrev = 0 AND bBoostPresEnable = 1
THEN
	TimerOn.IN := 0; (*Сбрасываем старт таймера*)
	bTimerOnStart := 1; (*Запускаем таймер*)
	TimerOn(IN := bTimerOnStart, PT := T#10S, Q => bTimerOnOut);
END_IF;

IF bBoostPresEnablePrev = 1 AND bBoostPresEnable = 0
THEN
	TimerOn.IN := 0; (*Сбрасываем старт таймера*)
END_IF;

IF rIW_BoostPres < 0.4 AND bBoostPresEnablePrev = 1 AND bTimerOnOut = 0
THEN
	bErrorNumber20       := 1;(**)
	dwHornEnable.20      := 0;(*Сирена отключена*)
	bLN2_WorkOverTemp    := 1;
	(*bQX_BoostPresEmergStop := 0;(*Останов работы центробежного насоса в режиме "Авто"*)*)
(*ELSIF rIW_BoostPres < 0.5 AND bBoostPresEnablePrev = 0
THEN
	bErrorNumber20       := 1;
	dwHornEnable.20      := 0;(*Сирена отключена*)*)
ELSE
	(*bErrorNumber20       := 0;*)
	dwHornEnable.20      := 0;
END_IF;

bBoostPresEnablePrev := bBoostPresEnable;

(*-----------------------------------------------------------------------------------------------------------------------------------------------------------------------------------*)
(*Формируем признак отключения автоматического режима при работе в режиме "Авто" при превышении температуры*)

IF byCurrStep = 3 AND rIW_LN2_Temp > rSet_LN2SaturTemp
THEN
	bLN2_WorkOverTemp := 1;
END_IF;

(*-----------------------------------------------------------------------------------------------------------------------------------------------------------------------------------*)
(**)

IF byCurrStep = 3 AND bIX_BlockOff = 1
THEN
	bLN2_WorkOverTemp := 1;
END_IF;

(*-----------------------------------------------------------------------------------------------------------------------------------------------------------------------------------*)
(*Отключаем ПИД в режиме "Ручной"*)

IF bBoostPresEnable = 0 (*Если переключен в режим "Ручной" извне переключателем или отключен с дисплея, то ПИД отключаем*)
THEN
	PID_3_Reset    := 1;
	rSet_BoostPres := 0;
	PID_3_Y_Manual := 1;
ELSE
	PID_3_Reset    := 0;
	PID_3_Y_Manual := 0;
END_IF;

(*-----------------------------------------------------------------------------------------------------------------------------------------------------------------------------------*)
(*ПИД-контур 2 поддержания давления нагнетания (подпитывающий насос)*)

PID_3(Actual      := rIW_BoostPres,
	Set_Point     := rSet_BoostPres,
	KP            := rArrayDataPID_P_Coef[3],
	TN            := rArrayDataPID_I_Coef[3],
	TV            := rArrayDataPID_D_Coef[3],
	Y_Manual      := PID_3_Y_Manual,
	Y_Offset      := rArrayDataPID_Shift[3],
	Y_Min         := rArrayDataPWM_YL[3],
	Y_Max         := rArrayDataPWM_YH[3] (*PID_3_Y_Max*),
	Manual        := PID_3_Manual,
	Reset         := PID_3_Reset,
	Y             => rPWM_BoostPres,
	Limits_Active => PID_3_Limits,
	Overflow      => PID_3_Overflow);

rArrayDataRAWPID[3] := rPWM_BoostPres;

(*-----------------------------------------------------------------------------------------------------------------------------------------------------------------------------------*)
(*Отключаемся от управления ШИМ в режиме "Ручной"*)

IF bBoostPresEnable = 0 (*Если переключен в режим "Ручной" извне переключателем или отключен с дисплея, то ШИМ отключаем*)
THEN
	rPWM_BoostPres := 0;
END_IF;

(*-----------------------------------------------------------------------------------------------------------------------------------------------------------------------------------*)
(*Обработка байта описания канала*)

CASE dwArrayDataPWM_DZ_MIN[3] OF
	0: rPWM_BoostPres := rPWM_BoostPres;
	1: rPWM_BoostPres := rArrayDataPWM_DZ_MAX[3];
	2: rPWM_BoostPres := rPWM_BoostPres * rArrayDataPWM_DZ_MAX[3];
	ELSE rPWM_BoostPres := rPWM_BoostPres;
END_CASE;

rArrayDataRAWPWM[3] := rPWM_BoostPres;

(*-----------------------------------------------------------------------------------------------------------------------------------------------------------------------------------*)
(*ШИМ-контроллер поддержания давления нагнетания (подпитывающий насос)*)

BoostPresFreqPWM(dwReriodPWM := dwArrayAverTimePWM[3], wFrequencyPWM => , bRestartPWM => );

PWM3(INIT := (bFirstIn OR BoostPresFreqPWM.bRestartPWM), FREQUENCY := BoostPresFreqPWM.wFrequencyPWM, CHANNEL := 2, VALUE := REAL_TO_WORD(rPWM_BoostPres), CHANGE := TRUE, DITHER_VALUE := 10, DITHER_FREQUENCY := 140);

(*-----------------------------------------------------------------------------------------------------------------------------------------------------------------------------------*)
(**)

bIX_BoostPresAutoModePrev := bIX_BoostPresAutoMode;

(*-----------------------------------------------------------------------------------------------------------------------------------------------------------------------------------*)
(*bErrorNumber18 - Ошибка 18. Центробеж. насос. Переведите регулятор в положение «0»*)
(*
IF byCurrStep = 3 AND bBoostPresEnable = 1 AND rPWM_BoostPres < 10
THEN
	bErrorNumber18  := 1;(*РАБОТАЕМ С ПРЕДУПРЕЖДЕНИЕМ*)
	dwHornEnable.18 := 0;(*Сирена отключена*)
ELSE
	bErrorNumber18  := 0;
	dwHornEnable.18 := 0;
END_IF;*)
END_PROGRAM

(* POU Output Modules/FREQ_CHANGE_PWM, ST *)
FUNCTION_BLOCK FREQ_CHANGE_PWM

VAR_INPUT
	dwReriodPWM     : DWORD;
END_VAR

VAR_OUTPUT
	wFrequencyPWM   : WORD;
	bRestartPWM     : BOOL;
END_VAR

VAR
	dwReriodPWMPrev : DWORD;
END_VAR
IF    dwReriodPWM = 0                       THEN wFrequencyPWM := 250;
ELSIF dwReriodPWM > 0 AND dwReriodPWM < 200 THEN wFrequencyPWM := 5000;
ELSIF dwReriodPWM > 100_000                 THEN wFrequencyPWM := 10;
ELSE  wFrequencyPWM := REAL_TO_WORD(1_000_000 / DWORD_TO_REAL(dwReriodPWM));
END_IF;

IF dwReriodPWM <> dwReriodPWMPrev
THEN
	bRestartPWM := 1;
ELSE
	bRestartPWM := 0;
END_IF;

dwReriodPWMPrev := dwReriodPWM;
END_FUNCTION_BLOCK

(* POU Output Modules/HydHeat_processing, ST *)
PROGRAM HydHeat_processing

VAR_INPUT
	bFirstIn                    : BOOL;
END_VAR

VAR
	bIX_HydHeatPresAutoModePrev : BOOL :=    0;
	bLN2_WorkOverTemp           : BOOL :=    0;

	bQX_HydHeatPresEmergStop    : BOOL :=    0;

	PID_1                       : PID;
 	PID_1_Reset                 : BOOL :=    0;
	PID_1_Limits                : BOOL :=    0;
	PID_1_Manual                : BOOL :=    0;
	PID_1_Y_Manual              : REAL :=    0;
	PID_1_Y_Max                 : REAL :=  500;
	PID_1_Overflow              : BOOL :=    0;

(*Переменные для канала ШИМ*)
	PWM1                        : PWM1000;(*Выход ШИМ канал 0 на пин 44*)
	HydHeatPresFreqPWM          : FREQ_CHANGE_PWM;
	rPWM_HydHeatPresPrev        : REAL;
	rHydHeatActualPoint         : REAL;
	rHydHeatSetPoint            : REAL;

	HydHeatRamp                  : RAMP_REAL;
	rHydHeatSetPointRampASCEND   : REAL :=     1;
	rHydHeatSetPointRampDESCEND  : REAL :=     1;
	rHydHeatSetPointRampTIMEBASE : TIME :=  T#1S;
END_VAR
(*-----------------------------------------------------------------------------------------------------------------------------------------------------------------------------------*)
(*Управляем давлением гидронагрева*)

bQX_HydHeatPresEmergStop := 1;(*Разрешаем работу гидронагрева (в режиме "Авто")*)

(*-----------------------------------------------------------------------------------------------------------------------------------------------------------------------------------*)
(*bErrorNumber19 - Ошибка 19. Гидронагрев. Температура жидкого азота выше допустимого*)
(*
IF rIW_LN2_Temp > rSet_LN2SaturTemp
THEN
	bErrorNumber19           := 1;(**)
	dwHornEnable.19          := 0;(*Сирена отключена*)
	(*bQX_HydHeatPresEmergStop := 0;(*Останов работы гидронагрева в режиме "Авто"*)*)
ELSE
	bErrorNumber19           := 0;
	dwHornEnable.19          := 0;
END_IF;
*)
(*-----------------------------------------------------------------------------------------------------------------------------------------------------------------------------------*)
(*bErrorNumber19 - 19. Гидронагрев. Обороты двигателя меньше допустимого*)

IF diCurrentEngineRPM < 1500
THEN
	bErrorNumber19           := 1;(**)
	dwHornEnable.19          := 0;(*Сирена отключена*)
	bQX_HydHeatPresEmergStop := 0;(*Останов работы гидронагрева в режиме "Авто"*)
ELSE
	bErrorNumber19           := 0;
	dwHornEnable.19          := 0;
END_IF;

(*-----------------------------------------------------------------------------------------------------------------------------------------------------------------------------------*)
(*bErrorNumber20 - Ошибка 20. Г/нагрев. Давление подпитки ниже допустимого*)
(*                 (*ПЕРЕНЕСЕНО В Boost_processing !!!!!!!!!!!!*)
IF rIW_BoostPres < 0.55
THEN
	bErrorNumber20           := 1;(**)
	dwHornEnable.20          := 0;(*Сирена отключена*)
	(*bQX_HydHeatPresEmergStop := 0;(*Останов работы гидронагрева в режиме "Авто"*)*)
ELSE
	bErrorNumber20           := 0;
	dwHornEnable.20          := 0;
END_IF;
*)

(*-----------------------------------------------------------------------------------------------------------------------------------------------------------------------------------*)
(*bErrorNumber21 - Ошибка 21. Гидронагрев. Температура ОЖ теплобменника ниже допустимого*)
(*
IF rIW_CoolTempIn < rCoolTempInMin
THEN
	bErrorNumber21           := 1;(**)
	dwHornEnable.21          := 0;(*Сирена отключена*)
	(*bQX_HydHeatPresEmergStop := 0;(*Останов работы гидронагрева в режиме "Авто"*)*)
ELSE
	bErrorNumber21           := 0;
	dwHornEnable.21          := 0;
END_IF;
*)
(*-----------------------------------------------------------------------------------------------------------------------------------------------------------------------------------*)
(*bErrorNumber22 - Ошибка 22. Гидронагрев. Скорость НВД меньше 20 об/мин*)
(*
IF rFRQ_TriplexRPM < 20
THEN
	bErrorNumber22           := 1;(**)
	dwHornEnable.22          := 0;(*Сирена отключена*)
	(*bQX_HydHeatPresEmergStop := 0;(*Останов работы гидронагрева в режиме "Авто"*)*)
ELSE
	bErrorNumber22           := 0;
	dwHornEnable.22          := 0;
END_IF;
*)
(*-----------------------------------------------------------------------------------------------------------------------------------------------------------------------------------*)
(*В итоге сформировали разрешение работы гидронагрева в режиме "Авто"*)

	(*bQX_HydHeatPresEmergStop = 1 - разрешаем работу гидронагрева в режиме "Авто"*)
	(*bQX_HydHeatPresEmergStop = 0 - блокируем работу гидронагрева в режиме "Авто"*)

(*-----------------------------------------------------------------------------------------------------------------------------------------------------------------------------------*)
(*Установка давления ? (температуры ?) гидронагрева после повторного возврата в режим "Авто"*)

IF bIX_HydHeatPresAutoModePrev = 0 AND bIX_HydHeatPresAutoMode = 1
THEN
	bLN2_WorkOverTemp := 0;
END_IF;

(*-----------------------------------------------------------------------------------------------------------------------------------------------------------------------------------*)
(*Формируем разрешение автоматического режима при положении тумблера "Авто"*)

IF byCurrStep = 3 AND bIX_HydHeatPresAutoMode = 1 AND bQX_HydHeatPresEmergStop = 1 AND bLN2_WorkOverTemp = 0 AND bIX_BlockOff = 0 AND bCommomErrorADC = 0
THEN
	bHydHeatPresEnable       := 1;
	rSet_GN2Temp             := rSet_GN2TempManual;
	bQX_HydHeatPresContrMode := 1;(*Зеленой лампочкой светим постоянно*)
ELSE
	bHydHeatPresEnable       := 0;
	bQX_HydHeatPresContrMode := 0;(*Зеленую лампочку погасили*)
END_IF;

(*-----------------------------------------------------------------------------------------------------------------------------------------------------------------------------------*)
(*Формируем признак отключенного автоматического режима при положении тумблера "Авто"*)

IF (*byCurrStep = 3 AND*) bIX_HydHeatPresAutoMode = 1 AND bHydHeatPresEnable = 0
THEN
	bHydHeatPresDisparity    := 1;
	bQX_HydHeatPresContrMode := bTimerBlinkOut;(*Зеленой лампочкой мигаем*)
ELSE
	bHydHeatPresDisparity    := 0;
END_IF;

(*-----------------------------------------------------------------------------------------------------------------------------------------------------------------------------------*)
(*Формируем признак отключения автоматического режима при работе в режиме "Авто" при включении аварийнго выхода из режима "Авто"*)

IF byCurrStep = 3 AND bQX_HydHeatPresEmergStop = 0
THEN
	bLN2_WorkOverTemp := 1;
END_IF;

(*-----------------------------------------------------------------------------------------------------------------------------------------------------------------------------------*)
(**)

IF byCurrStep = 3 AND bIX_BlockOff = 1
THEN
	bLN2_WorkOverTemp := 1;
END_IF;

(*-----------------------------------------------------------------------------------------------------------------------------------------------------------------------------------*)
(*Отключаем ПИД в режиме "Ручной"*)

IF bIX_HydHeatPresAutoMode = 0 OR bHydHeatPresEnable  = 0 (*Если переключен в режим "Ручной" извне переключателем, то ПИД отключаем*)
THEN
	PID_1_Reset    := 1;
	rSet_GN2Temp   := 0;
	PID_1_Y_Manual := 1;
ELSE
	PID_1_Reset    := 0;
	PID_1_Y_Manual := 0;
END_IF;

(*-----------------------------------------------------------------------------------------------------------------------------------------------------------------------------------*)
(**)

IF (*bTriplexRPMEnable = 1*) rFRQ_TriplexRPM > 10
THEN
	rHydHeatActualPoint := rIW_GN2_Temp;
	PID_1_Y_Max := rArrayDataPWM_YH[1];
	rHydHeatSetPoint := rSet_GN2Temp;
ELSE
	rHydHeatActualPoint := rIW_CoolTempIn;
	PID_1_Y_Max := 0.3 * rArrayDataPWM_YH[1];
	rHydHeatSetPoint := rCoolTempInMin;
END_IF;

(*-----------------------------------------------------------------------------------------------------------------------------------------------------------------------------------*)
(*ПИД-контур 2 поддержания давления гидронагрева*)

HydHeatRamp(
			IN       := rHydHeatSetPoint,
			ASCEND   := rHydHeatSetPointRampASCEND,
			DESCEND  := rHydHeatSetPointRampDESCEND,
			TIMEBASE := rHydHeatSetPointRampTIMEBASE,
			RESET    := 0,
			OUT      => );

PID_1(Actual      := rHydHeatActualPoint,
	Set_Point     := HydHeatRamp.OUT (*rHydHeatSetPoint*),
	KP            := rArrayDataPID_P_Coef[1],
	TN            := rArrayDataPID_I_Coef[1],
	TV            := rArrayDataPID_D_Coef[1],
	Y_Manual      := PID_1_Y_Manual,
	Y_Offset      := rArrayDataPID_Shift[1],
	Y_Min         := rArrayDataPWM_YL[1],
	Y_Max         := PID_1_Y_Max,
	Manual        := PID_1_Manual,
	Reset         := PID_1_Reset,
	Y             => rPWM_HydHeatPres,
	Limits_Active => PID_1_Limits,
	Overflow      => PID_1_Overflow);

rArrayDataRAWPID[1] := rPWM_HydHeatPres;

(*-----------------------------------------------------------------------------------------------------------------------------------------------------------------------------------*)
(*Ограничиваем выходное значение ШИМ при достижении давления 350 Бар*)

(*IF rIW_HydHeatPres > 35
THEN
	rPWM_HydHeatPres := rPWM_HydHeatPresPrev;
	PID_1_Manual     := 1;
	PID_1_Y_Manual   := rPWM_HydHeatPresPrev;
ELSE
	PID_1_Manual     := 0;
END_IF;

rPWM_HydHeatPresPrev := rPWM_HydHeatPres;*)

(*-----------------------------------------------------------------------------------------------------------------------------------------------------------------------------------*)
(*Отключаемся от управления ШИМ в режиме "Ручной"*)

IF bIX_HydHeatPresAutoMode = 0 OR bHydHeatPresEnable  = 0 (*Если переключен в режим "Ручной" извне переключателем, то ШИМ отключаем*)
THEN
	rPWM_HydHeatPres := 0;
END_IF;

(*-----------------------------------------------------------------------------------------------------------------------------------------------------------------------------------*)
(*Обработка байта описания канала*)

CASE dwArrayDataPWM_DZ_MIN[1] OF
	0: rPWM_HydHeatPres := rPWM_HydHeatPres;
	1: rPWM_HydHeatPres := rArrayDataPWM_DZ_MAX[1];
	2: rPWM_HydHeatPres := rPWM_HydHeatPres * rArrayDataPWM_DZ_MAX[1];
	ELSE rPWM_HydHeatPres := rPWM_HydHeatPres;
END_CASE;

rArrayDataRAWPWM[1] := rPWM_HydHeatPres;

(*-----------------------------------------------------------------------------------------------------------------------------------------------------------------------------------*)
(*ШИМ-контроллер поддержания давления гидронагрева*)

HydHeatPresFreqPWM(dwReriodPWM := dwArrayAverTimePWM[1], wFrequencyPWM => , bRestartPWM => );

PWM1(INIT := (bFirstIn OR HydHeatPresFreqPWM.bRestartPWM), FREQUENCY := HydHeatPresFreqPWM.wFrequencyPWM, CHANNEL := 0, VALUE:=REAL_TO_WORD(rPWM_HydHeatPres), CHANGE := TRUE, DITHER_VALUE := 10, DITHER_FREQUENCY := 140);

(*-----------------------------------------------------------------------------------------------------------------------------------------------------------------------------------*)
(**)

bIX_HydHeatPresAutoModePrev := bIX_HydHeatPresAutoMode;

(*-----------------------------------------------------------------------------------------------------------------------------------------------------------------------------------*)
(*Расчет рассогласования расчетной и текущей величины*)

rHydHeatPres_Calc := HydHeatPres_calculation(rPWMcurr := (rPWM_HydHeatPres / 10));

IF rIW_HydHeatPres > 0.01
THEN
	rHydHeatPres_Err := (rHydHeatPres_Calc - rIW_HydHeatPres) * 100 / rIW_HydHeatPres;
ELSE
	rHydHeatPres_Err := 0;
END_IF;

(*-----------------------------------------------------------------------------------------------------------------------------------------------------------------------------------*)
(*bErrorNumber23 - Ошибка 23. Гидронагрев. Переведите регулятор в положение «0»*)
(*
IF byCurrStep = 3 AND bHydHeatPresEnable = 1 AND (*ABS(rHydHeatPres_Err) > 20*) rPWM_HydHeatPres < 100 AND rIW_HydHeatPres > 1.5
THEN
	bErrorNumber23  := 1;(*РАБОТАЕМ С ПРЕДУПРЕЖДЕНИЕМ*)
	dwHornEnable.23 := 0;(*Сирена отключена*)
ELSE
	bErrorNumber23  := 0;
	dwHornEnable.23 := 0;
END_IF;*)
END_PROGRAM

(* POU Service/HydHeatPres_calculation, ST *)
FUNCTION HydHeatPres_calculation : REAL

VAR_INPUT
	rPWMcurr : REAL;(*Текущее значение ШИМ, %*)
END_VAR

VAR
END_VAR
(*-----------------------------------------------------------------------------------------------------------------------------------------------------------------------------------*)
(**)

HydHeatPres_calculation := (9 + 6.686 * rPWMcurr) / 10;(*Формула в бар, поэтому делим на 10*)
END_FUNCTION

(* POU Output Modules/Triplex_processing, ST *)
PROGRAM Triplex_processing

VAR_INPUT
	bFirstIn                   : BOOL;
END_VAR

VAR
	bIX_TriplexRPMAutoModePrev : BOOL :=    0;
	bLN2_WorkOverTemp          : BOOL :=    0;

	PID_2                      : PID;
 	PID_2_Reset                : BOOL :=    0;
	PID_2_Limits               : BOOL :=    0;
	PID_2_Manual               : BOOL :=    0;
	PID_2_Y_Manual             : REAL :=    0;
	PID_2_Y_Max                : REAL :=  400 (*1000*);
	PID_2_Overflow             : BOOL :=    0;

(*Переменные для канала ШИМ*)
	PWM2                       : PWM1000;(*Выход ШИМ канал 1 на пин 45*)
	TriplexRPMFreqPWM          : FREQ_CHANGE_PWM;

	bBlockDisablePrev          : BOOL;
	bTriplexRPMEnablePrev      : BOOL;

	bTriplexRPMState           : BOOL;(*Контроль состояния НВД, работает или нет, в текущем цикле*)
	bTriplexRPMStatePrev       : BOOL;(*Контроль состояния НВД, работает или нет, в предыдущем цикле*)
END_VAR
(*-----------------------------------------------------------------------------------------------------------------------------------------------------------------------------------*)
(*Определяем предыдущее и текущее состояние НВД, независимо, ручной или автоматический режим работы*)

IF rFRQ_TriplexRPM > 1
THEN
	bTriplexRPMState := 1;
ELSE
	bTriplexRPMState := 0;
END_IF;

bTriplexRPMStatePrev := bTriplexRPMState;

(*-----------------------------------------------------------------------------------------------------------------------------------------------------------------------------------*)
(*Расчет минимальной температуры теплообменника*)

rCoolTempInMin := Temperature_calculation(  rTmin := rSet_GN2TempManual (*37.8*),
											rVreq := rSet_GN2Rate,
											rPprs := rIW_GN2_Pres,
											rTreq := rSet_GN2TempManual,
											rK    := 1.5 (*2.56*));

(*-----------------------------------------------------------------------------------------------------------------------------------------------------------------------------------*)
(*Расчет количества оборотов НВД исходя из требуемого расхода*)

rSet_TriplexRPMManual := rSet_GN2Rate / 0.08786324786325;

(*-----------------------------------------------------------------------------------------------------------------------------------------------------------------------------------*)
(*Управляем оборотами НВД*)

IF byCurrStep = 3
THEN
	bQX_TriplexEmergStop := 1;(*Разрешаем работу НВД*)
ELSE
	bQX_TriplexEmergStop := 0;(*Запрещаем работу НВД*)
END_IF

(*-----------------------------------------------------------------------------------------------------------------------------------------------------------------------------------*)
(*Ошибка 04. Давление  газообр. азота выше допустимого*)

IF rIW_GN2_Pres > rSet_GN2OverPres AND (byCurrStep = 1 OR byCurrStep = 2 OR byCurrStep = 3 OR byCurrStep = 4)
THEN
	bErrorNumber04       := 1;
	dwHornEnable.4       := 1;(*Сирена включена*)
	bQX_TriplexEmergStop := 0;(*Останов НВД*)
ELSE
	(*bErrorNumber04       := 0;*)
	dwHornEnable.4       := 0;
END_IF;

(*-----------------------------------------------------------------------------------------------------------------------------------------------------------------------------------*)
(*bErrorNumber08 - Ошибка 08. НВД. Температура жидкого азота выше допустимого*)  (*КРАСНЫЙ !!!!!!!!!!!!!!!!!!!*)

IF (byCurrStep = 3 OR byCurrStep = 4) AND rIW_LN2_Temp > rSet_LN2SaturTempTriplex AND bTriplexRPMStatePrev = 1
THEN
	bErrorNumber08       := 1;
	dwHornEnable.8       := 0;(*Сирена отключена*)
	bQX_TriplexEmergStop := 0;(*Останов НВД*)
ELSE
	(*bErrorNumber08       := 0;*)
	dwHornEnable.8       := 0;
END_IF;

(*-----------------------------------------------------------------------------------------------------------------------------------------------------------------------------------*)
(*bErrorNumber09 - Ошибка 09. НВД. Давление подпитки ниже допустимого*)  (*КРАСНЫЙ !!!!!!!!!!!!!!!!!!!*)

IF (byCurrStep = 3 OR byCurrStep = 4) AND rIW_BoostPres < 0.45 AND bTriplexRPMStatePrev = 1
THEN
	bErrorNumber09       := 1;
	dwHornEnable.9       := 0;(*Сирена отключена*)
	bQX_TriplexEmergStop := 0;(*Останов НВД*)
ELSE
	(*bErrorNumber09       := 0;*)
	dwHornEnable.9       := 0;
END_IF;

(*-----------------------------------------------------------------------------------------------------------------------------------------------------------------------------------*)
(*bErrorNumber13 - Ошибка 13. НВД.Температура жидкого азота выше допустимого*) (*ЖЕЛТЫЙ !!!!!!!!!!!!!!!!!!!*)

IF (*(byCurrStep = 0 OR byCurrStep = 1 OR byCurrStep = 2) AND*) rIW_LN2_Temp > rSet_LN2SaturTempTriplex AND bTriplexRPMStatePrev = 0
THEN
	bErrorNumber13       := 1;
	dwHornEnable.13      := 0;(*Сирена отключена*)
	bQX_TriplexEmergStop := 0;(*Останов НВД*)
ELSE
	(*bErrorNumber13       := 0;*)
	dwHornEnable.13      := 0;
END_IF;

(*-----------------------------------------------------------------------------------------------------------------------------------------------------------------------------------*)
(*bErrorNumber14 - Ошибка 14. НВД. Давление подпитки ниже допустимого*) (*ЖЕЛТЫЙ !!!!!!!!!!!!!!!!!!!*)

IF (*(byCurrStep = 0 OR byCurrStep = 1 OR byCurrStep = 2) AND*) rIW_BoostPres < 0.45  AND bTriplexRPMStatePrev = 0
THEN
	bErrorNumber14       := 1;
	dwHornEnable.14      := 0;(*Сирена отключена*)
	bQX_TriplexEmergStop := 0;(*Останов НВД*)
ELSE
	(*bErrorNumber14       := 0;*)
	dwHornEnable.14      := 0;
END_IF;

(*-----------------------------------------------------------------------------------------------------------------------------------------------------------------------------------*)
(*bErrorNumber15 - Ошибка 15. НВД. Температура ОЖ теплобменника ниже допустимого*)
(*                        (*ПЕРЕНЕСЕНО НИЖЕ !!!!!!!!!!!!*)
IF rIW_CoolTempIn < rCoolTempInMin AND bTriplexRPMEnable = 1
THEN
	bErrorNumber15       := 1;
	dwHornEnable.15      := 0;(*Сирена отключена*)
ELSIF rIW_CoolTempIn < rCoolTempInMin AND bTriplexRPMEnable = 0
THEN
	bErrorNumber15       := 1;
	dwHornEnable.15      := 0;(*Сирена отключена*)
	bLN2_WorkOverTemp    := 1;
ELSE
	bErrorNumber15       := 0;
	dwHornEnable.15      := 0;
END_IF;
*)

(*-----------------------------------------------------------------------------------------------------------------------------------------------------------------------------------*)
(*Разрешаем вращение НВД при нажатии разблокирующей кнопки и оборотах меньше 20 об/мин*)

IF bBlockDisable = 1 AND rFRQ_TriplexRPM < 20
THEN
	bQX_TriplexEmergStop := 1;(*Разрешаем вращение НВД*)
	IF bBlockDisablePrev = 0 AND bBlockDisable = 1
	THEN bResetErrors := 1;
	END_IF;
END_IF;

bBlockDisablePrev := bBlockDisable;

(*-----------------------------------------------------------------------------------------------------------------------------------------------------------------------------------*)
(*В итоге сформировали разрешение работы НВД (независимо от положении тумблера "Ручной"/"Авто")*)

	(*bQX_TriplexEmergStop = 1 - разрешаем вращение НВД*)
	(*bQX_TriplexEmergStop = 0 - блокируем вращение НВД*)

(*-----------------------------------------------------------------------------------------------------------------------------------------------------------------------------------*)
(*Установка оборотов НВД после повторного возврата в режим "Авто"*)

IF bIX_TriplexRPMAutoModePrev = 0 AND bIX_TriplexRPMAutoMode = 1
THEN
	bLN2_WorkOverTemp := 0;
END_IF;

(*-----------------------------------------------------------------------------------------------------------------------------------------------------------------------------------*)
(*Формируем разрешение автоматического режима при положении тумблера "Авто"*)

IF byCurrStep = 3 AND bIX_TriplexRPMAutoMode = 1 AND bQX_TriplexEmergStopTrig (*bQX_TriplexEmergStop*) = 1 AND bLN2_WorkOverTemp = 0 AND bIX_BlockOff = 0 AND bCommomErrorADC = 0
THEN
	bTriplexRPMEnable       := 1;
	rSet_TriplexRPM         := rSet_TriplexRPMManual;
	bQX_TriplexRPMContrMode := 1;(*Зеленой лампочкой светим постоянно*)
ELSE
	bTriplexRPMEnable       := 0;
	bQX_TriplexRPMContrMode := 0;(*Зеленую лампочку погасили*)
END_IF;

(*-----------------------------------------------------------------------------------------------------------------------------------------------------------------------------------*)
(*Формируем признак отключенного автоматического режима при положении тумблера "Авто"*)

IF (*byCurrStep = 3 AND*) bIX_TriplexRPMAutoMode = 1 AND bTriplexRPMEnable = 0 THEN
	bTriplexRPMDisparity    := 1;
	bQX_TriplexRPMContrMode := bTimerBlinkOut;(*Зеленой лампочкой мигаем*)
ELSE
	bTriplexRPMDisparity    := 0;
END_IF;

(*-----------------------------------------------------------------------------------------------------------------------------------------------------------------------------------*)
(*bErrorNumber15 - Ошибка 15. НВД. Температура ОЖ теплобменника ниже допустимого*)

IF rIW_CoolTempIn < rCoolTempInMin AND bTriplexRPMEnablePrev = 1
THEN
	bErrorNumber15       := 0;(*Предупреждение решили НЕ давать*)
	dwHornEnable.15      := 0;(*Сирена отключена*)
ELSIF rIW_CoolTempIn < rCoolTempInMin AND bTriplexRPMEnablePrev = 0
THEN
	bErrorNumber15       := 1;
	dwHornEnable.15      := 0;(*Сирена отключена*)
	bLN2_WorkOverTemp    := 1;
ELSE
	bErrorNumber15       := 0;
	dwHornEnable.15      := 0;
END_IF;

bTriplexRPMEnablePrev := bTriplexRPMEnable;

(*-----------------------------------------------------------------------------------------------------------------------------------------------------------------------------------*)
(*Формируем признак отключения автоматического режима при работе в режиме "Авто" при включении аварийной блокировки*)

IF byCurrStep = 3 AND bQX_TriplexEmergStop = 0 THEN
	bLN2_WorkOverTemp := 1;
END_IF;

(*-----------------------------------------------------------------------------------------------------------------------------------------------------------------------------------*)
(**)

IF byCurrStep = 3 AND bIX_BlockOff = 1
THEN
	bLN2_WorkOverTemp := 1;
END_IF;

(*-----------------------------------------------------------------------------------------------------------------------------------------------------------------------------------*)
(*Отключаем ПИД в режиме "Ручной"*)

